                        #IEC_Timer.Spülen(IN := #Zst."TON_CM05.QM62_auf" AND #Out.QM63,
                                          PT := #Param.Spülzeit,
                                          Q => #Zst.Spuelen,
                                          ET => #Spülzeit);
                        #Zst.Restzeit_Spülen := #Param.Spülzeit - #Spülzeit;

                        IF #Zst."TON_CM05.QM62_auf" AND #Out.QM63 AND #In."SRM_CM05.QM61_zu" AND #In."SRM_CM05.QM64_zu" AND NOT #Zst.Spuelen THEN
                            #Zst.Spuelen_aktiv := FALSE;
                            #Out.QM62 := FALSE;
                        END_IF;

                        // Fertig
                        IF NOT #Zst.Spuelen AND NOT #Zst.Spuelen_aktiv AND NOT #Out.QM63 THEN
                            #Out.QM62 := #Out.QM63 := FALSE;
                            #Zst.Restzeit_Spülen := T#0s;
                            #Mld.Pu_Spuelen_Fertig := TRUE;
                        END_IF;
                    ELSE
                        #Out.QM62 := FALSE;
                        #Out.QM63 := FALSE;
                        #Zst.Restzeit_Spülen := T#0s;
                    END_IF;
                    #Out.GP11_Ein := FALSE;

           2: // Spülen + Drucktest - nur Hand
               // Ventile Abpumpen zu    
               #Out.QM61 := FALSE;
               #Out.QM64 := FALSE;
               IF NOT #Zst.Drucktest_aktiv THEN
                   IF #In.Ein THEN
                       IF #posFl_Hand THEN
                           #Zst.Spuelen_aktiv := TRUE;
                       END_IF;
                       #Out.QM62 := NOT #In."Niv_max_CM05.BL01" AND NOT #In."Niv_Uel_CM05.BL05";
                       #Out.QM63 := #Out.QM62;
                       #IEC_Timer.Spülen(IN := #Zst."TON_CM05.QM62_auf" AND #Out.QM63 AND #In."SRM_CM05.QM61_zu" AND #In."SRM_CM05.QM64_zu",
                                         PT := #Param.Spülzeit,
                                         Q => #Zst.Spuelen,
                                         ET => #Spülzeit);
                       #Zst.Restzeit_Spülen := #Param.Spülzeit - #Spülzeit;

                       IF #Zst."TON_CM05.QM62_auf" AND #Out.QM63 AND #In."SRM_CM05.QM61_zu" AND #In."SRM_CM05.QM64_zu" AND NOT #Zst.Spuelen THEN
                           #Zst.Spuelen_aktiv := FALSE;
                       END_IF;

                       // Fertig
                       IF NOT #Zst.Spuelen AND NOT #Zst.Spuelen_aktiv THEN
                           #Out.QM62 := #Out.QM63 := FALSE;
                           #Zst.Restzeit_Spülen := T#0s;
                           #Zst.Drucktest_aktiv := TRUE;
                           #Zst.Status_DT := #S1;
                       END_IF;
                   ELSE
                       #Out.QM62 := FALSE;
                       #Out.QM63 := FALSE;
                       #Zst.Restzeit_Spülen := T#0s;
                   END_IF;
                   #Out.GP11_Ein := FALSE;
               END_IF;

               IF #Zst.Drucktest_aktiv THEN
                   CASE #Zst.Status_DT OF
                       #S1:  //Druckaufbau

                           IF "DB_Temporaer".Drucksensoren_deaktiviert THEN
                               #Zst.Drucktest_ok := TRUE;

                               "Ergebnis_DT"("Name" := #"Name",
                                             akt_Zeit := "Uhrzeit".aktDatum,
                                             ok := #Zst.Drucktest_ok,
                                             Fehler := NOT #Zst.Drucktest_ok);

                               #Mld.Drucktest_ok := #Zst.Drucktest_ok;
                               #Mld.DT_Fehler := NOT #Zst.Drucktest_ok;
                               #Zst.Status_DT := #S4;
                           ELSE
                               #Out.QM62 := TRUE;
                               IF (#In.Druck_Pumpe > #Param.SW_Drucktest + 0.25) OR #Mld.TO_Druckaufbau THEN
                                   #Zst.Status_DT := #S2;
                               END_IF;
                               #Zst.Restzeit_DT := #Param.DT_Druckaufbau - #IEC_Timer.TO_Druckaufbau.ET;
                           END_IF;

                       #S2: //Wartezeit
                           #IEC_Timer.Drucktest(IN := NOT #Out.QM62,
                                                PT := #Param.DT_Testzeit,
                                                Q => #Zst.Zeit_laeuft,
                                                ET => #Zeit_DT);
                           #Zst.Restzeit_DT := #Param.DT_Testzeit - #Zeit_DT;

                           IF NOT #Zst.Zeit_laeuft AND NOT #Out.QM62 THEN
                               #Zst.Restzeit_DT := T#0s;
                               #Zst.Status_DT := #S3;
                           END_IF;
                           #Out.QM62 := FALSE;

                       #S3:// Überprüfung
                           #Zst.Drucktest_ok := #In.Druck_Pumpe >= #Param.SW_Drucktest;

                           "Ergebnis_DT"("Name" := #"Name",
                                         akt_Zeit := "Uhrzeit".aktDatum,
                                         ok := #Zst.Drucktest_ok,
                                         Fehler := NOT #Zst.Drucktest_ok);

                           #Mld.Drucktest_ok := #Zst.Drucktest_ok;
                           #Mld.DT_Fehler := NOT #Zst.Drucktest_ok;
                           #Zst.Status_DT := #S4;

                       #S4: // Ende
                           ;
                   END_CASE;
               END_IF;
       END_CASE;
   ELSE
       #Out.GP11_Ein := FALSE;
       #Out.QM61 := FALSE;
       #Out.QM62 := FALSE;
       #Out.QM63 := FALSE;
       #Out.QM64 := FALSE;
   END_IF;
END_REGION

REGION Network 3 (SCL): Überwachung / Meldungen
   // Motorschutzschalter
   #Mld.MSS := NOT #In.MSS_ok AND NOT #In.NotHalt;
   // Trockenlaufschutz
   #Mld."TLS_CM05.BL03" := NOT #In."Niv_TLS_CM05.BL03";
   // Überlauf
   #Mld."Uel_CM05.BL05" := #In."Niv_Uel_CM05.BL05";
   // AWA nicht betriebsbereit
   #Mld.AWA_niO := NOT #In.AWA_ok;
   // keine Freigabe Abpumpen
   #Mld.keine_Frg_AWA := NOT #In.Frg_AWA;

   // Zeitüberschreitung Druckaufbau
   #IEC_Timer.TO_Druckaufbau(IN := #Zst.Status_DT = #S1,
                             PT := #Param.DT_Druckaufbau,
                             Q => #Mld.TO_Druckaufbau);

   // Grenzwert Pumpendruck
   #IEC_Timer.GW_p(IN := #Out.GP11_Ein,
                   PT := T#3s,
                   Q => #GP11_Laeuft);

   #Mld.GW_p := #GP11_Laeuft AND #In.GW_p;
   // nicht in Automatik
   #Mld.n_Auto := NOT #In.Auto AND "DB_ANLAGE".BA.Automat_ein;
END_REGION

REGION Network 4 (SCL): --> Visu
   // Status Pumpe
   "Status_E0A"(Hand := #In.Ein,
                Auto := #In.Auto,
                SonderModus_PumpeSpuelen:=#Zst.Spuelen,
                Stoerung := NOT #In.MSS_ok,
                Ausgang := #Out.GP11_Ein,
                StatusByte => #Zst.Status_GP11);
   // Anzeige Füllstand
   "Niv_Visu"(Niv_1 := #In."Niv_TLS_CM05.BL03",
              Niv_2 := #In."Niv_min_CM05.BL02",
              Niv_3 := #In."Niv_max_CM05.BL01",
              Niv_4 := #In."Niv_Uel_CM05.BL05",
              Niv_5 := FALSE,
              Niv_6 := FALSE,
              Wert_1 := #Niv_TLS,
              Wert_2 := #Niv_Min,
              Wert_3 := #Niv_max,
              Wert_4 := #Niv_Uel,
              Wert_5 := 0,
              Wert_6 := 0,
              Niveau => #Zst.Niveau,
              Niv_Err => #Mld.Niv_Sensorfehler);
END_REGION
END_FUNCTION_BLOCK

FUNCTION_BLOCK "Ventil_Stati"   // FB1095, LAD
TITLE = Ventilstatus
{ S7_Optimized_Access := 'TRUE' }
// 0: geschlossen (grau)
// 1: geöffnet (grün)
// 2: Störung (rot)
// stored: AutoNumber false, MemoryReserve 100, SetENOAutomatically false
   VAR RETAIN
      Param { ExternalAccessible := 'False'; ExternalVisible := 'False'; ExternalWritable := 'False'} : Struct
         "TO" : Time := T#20s;
      END_STRUCT;
      Mld : Struct
         "TO_auf_CM01.QM18" : Bool;
         "TO_zu_CM01.QM18" : Bool;
         "SF_CM01.QM18" : Bool;
         "TO_auf_CM01.QM19" : Bool;
         "TO_zu_CM01.QM19" : Bool;
         "SF_CM01.QM19" : Bool;
         "TO_auf_CM01.QM20" : Bool;
         "TO_zu_CM01.QM20" : Bool;
         "SF_CM01.QM20" : Bool;
         "TO_auf_CM01.QM25" : Bool;
         "TO_zu_CM01.QM25" : Bool;
         "SF_CM01.QM25" : Bool;
         "TO_auf_CM01.QM26" : Bool;
         "TO_zu_CM01.QM26" : Bool;
         "SF_CM01.QM26" : Bool;
         "TO_auf_CM01.QM27" : Bool;
         "TO_zu_CM01.QM27" : Bool;
         "SF_CM01.QM27" : Bool;
         "TO_auf_CM02.QM55" : Bool;
         "TO_zu_CM02.QM55" : Bool;
         "SF_CM02.QM55" : Bool;
         "TO_auf_CM02.QM56" : Bool;
         "TO_zu_CM02.QM56" : Bool;
         "SF_CM02.QM56" : Bool;
         "TO_auf_CM02.QM57" : Bool;
         "TO_zu_CM02.QM57" : Bool;
         "SF_CM02.QM57" : Bool;
         "TO_auf_CM02.QM62" : Bool;
         "TO_zu_CM02.QM62" : Bool;
         "SF_CM02.QM62" : Bool;
         "TO_auf_CM02.QM63" : Bool;
         "TO_zu_CM02.QM63" : Bool;
         "SF_CM02.QM63" : Bool;
         "TO_auf_CM02.QM64" : Bool;
         "TO_zu_CM02.QM64" : Bool;
         "SF_CM02.QM64" : Bool;
         "TO_auf_HQ01.QM21" : Bool;
         "TO_zu_HQ01.QM21" : Bool;
         "SF_HQ01.QM21" : Bool;
         "TO_auf_HQ01.QM22" : Bool;
         "TO_zu_HQ01.QM22" : Bool;
         "SF_HQ01.QM22" : Bool;
         "TO_auf_HQ01.QM23" : Bool;
         "TO_zu_HQ01.QM23" : Bool;
         "SF_HQ01.QM23" : Bool;
         "TO_auf_HQ01.QM24" : Bool;
         "TO_zu_HQ01.QM24" : Bool;
         "SF_HQ01.QM24" : Bool;
         "TO_auf_HQ01.LV01" : Bool;
         "TO_zu_HQ01.LV01" : Bool;
         "SF_HQ01.LV01" : Bool;
         "TO_auf_HQ02.QM58" : Bool;
         "TO_zu_HQ02.QM58" : Bool;
         "SF_HQ02.QM58" : Bool;
         "TO_auf_HQ02.QM59" : Bool;
         "TO_zu_HQ02.QM59" : Bool;
         "SF_HQ02.QM59" : Bool;
         "TO_auf_HQ02.QM60" : Bool;
         "TO_zu_HQ02.QM60" : Bool;
         "SF_HQ02.QM60" : Bool;
         "TO_auf_HQ02.QM61" : Bool;
         "TO_zu_HQ02.QM61" : Bool;
         "SF_HQ02.QM61" : Bool;
         "TO_auf_HQ02.LV02" : Bool;
         "TO_zu_HQ02.LV02" : Bool;
         "SF_HQ02.LV02" : Bool;
         "TO_auf_CM03.QM33" : Bool;
         "TO_zu_CM03.QM33" : Bool;
         "SF_CM03.QM33" : Bool;
         "TO_auf_CM03.QM34" : Bool;
         "TO_zu_CM03.QM34" : Bool;
         "SF_CM03.QM34" : Bool;
         "TO_auf_CM04.QM72" : Bool;
         "TO_zu_CM04.QM72" : Bool;
         "SF_CM04.QM72" : Bool;
         "TO_auf_CM04.QM73" : Bool;
         "TO_zu_CM04.QM73" : Bool;
         "SF_CM04.QM73" : Bool;
         "TO_auf_CM05.QM61" : Bool;
         "TO_zu_CM05.QM61" : Bool;
         "SF_CM05.QM61" : Bool;
         "TO_auf_CM05.QM64" : Bool;
         "TO_zu_CM05.QM64" : Bool;
         "SF_CM05.QM64" : Bool;
         "TO_auf_GP01.QM14" : Bool;
         "TO_zu_GP01.QM14" : Bool;
         "SF_GP01.QM14" : Bool;
         "TO_auf_GP01.QM15" : Bool;
         "TO_zu_GP01.QM15" : Bool;
         "SF_GP01.QM15" : Bool;
         "TO_auf_GP01.QM16" : Bool;
         "TO_zu_GP01.QM16" : Bool;
         "SF_GP01.QM16" : Bool;
         "TO_auf_GP01.QM17" : Bool;
         "TO_zu_GP01.QM17" : Bool;
         "SF_GP01.QM17" : Bool;
         "TO_auf_GP01.QM18" : Bool;
         "TO_zu_GP01.QM18" : Bool;
         "SF_GP01.QM18" : Bool;
         "TO_auf_GP01.QM19" : Bool;
         "TO_zu_GP01.QM19" : Bool;
         "SF_GP01.QM19" : Bool;
         "TO_auf_GP01.QM20" : Bool;
         "TO_zu_GP01.QM20" : Bool;
         "SF_GP01.QM20" : Bool;
         "TO_auf_GP01.QM21" : Bool;
         "TO_zu_GP01.QM21" : Bool;
         "SF_GP01.QM21" : Bool;
         "TO_auf_GP01.QM22" : Bool;
         "TO_zu_GP01.QM22" : Bool;
         "SF_GP01.QM22" : Bool;
         "TO_auf_GP02.QM38" : Bool;
         "TO_zu_GP02.QM38" : Bool;
         "SF_GP02.QM38" : Bool;
         "TO_auf_GP02.QM39" : Bool;
         "TO_zu_GP02.QM39" : Bool;
         "SF_GP02.QM39" : Bool;
         "TO_auf_GP02.QM40" : Bool;
         "TO_zu_GP02.QM40" : Bool;
         "SF_GP02.QM40" : Bool;
         "TO_auf_GP02.QM41" : Bool;
         "TO_zu_GP02.QM41" : Bool;
         "SF_GP02.QM41" : Bool;
         "TO_auf_GP02.QM42" : Bool;
         "TO_zu_GP02.QM42" : Bool;
         "SF_GP02.QM42" : Bool;
         "TO_auf_GP02.QM43" : Bool;
         "TO_zu_GP02.QM43" : Bool;
         "SF_GP02.QM43" : Bool;
         "TO_auf_GP02.QM44" : Bool;
         "TO_zu_GP02.QM44" : Bool;
         "SF_GP02.QM44" : Bool;
         "TO_auf_GP02.QM45" : Bool;
         "TO_zu_GP02.QM45" : Bool;
         "SF_GP02.QM45" : Bool;
         "TO_auf_GP02.QM46" : Bool;
         "TO_zu_GP02.QM46" : Bool;
         "SF_GP02.QM46" : Bool;
      END_STRUCT;
   END_VAR
   VAR
      IEC_Timer { ExternalAccessible := 'False'; ExternalVisible := 'False'; ExternalWritable := 'False'} : Struct
         "TO_auf_CM01.QM18" { S7_SetPoint := 'True'} : TON_TIME;
         "TO_zu_CM01.QM18" { S7_SetPoint := 'True'} : TON_TIME;
         "TO_auf_CM01.QM19" { S7_SetPoint := 'True'} : TON_TIME;
         "TO_zu_CM01.QM19" { S7_SetPoint := 'True'} : TON_TIME;
         "TO_auf_CM01.QM20" { S7_SetPoint := 'True'} : TON_TIME;
         "TO_zu_CM01.QM20" { S7_SetPoint := 'True'} : TON_TIME;
         "TO_auf_CM01.QM25" { S7_SetPoint := 'True'} : TON_TIME;
         "TO_zu_CM01.QM25" { S7_SetPoint := 'True'} : TON_TIME;
         "TO_auf_CM01.QM26" { S7_SetPoint := 'True'} : TON_TIME;
         "TO_zu_CM01.QM26" { S7_SetPoint := 'True'} : TON_TIME;
         "TO_auf_CM01.QM27" { S7_SetPoint := 'True'} : TON_TIME;
         "TO_zu_CM01.QM27" { S7_SetPoint := 'True'} : TON_TIME;
         "TO_auf_CM02.QM55" { S7_SetPoint := 'True'} : TON_TIME;
         "TO_zu_CM02.QM55" { S7_SetPoint := 'True'} : TON_TIME;
         "TO_auf_CM02.QM56" { S7_SetPoint := 'True'} : TON_TIME;
         "TO_zu_CM02.QM56" { S7_SetPoint := 'True'} : TON_TIME;
         "TO_auf_CM02.QM57" { S7_SetPoint := 'True'} : TON_TIME;
         "TO_zu_CM02.QM57" { S7_SetPoint := 'True'} : TON_TIME;
         "TO_auf_CM02.QM62" { S7_SetPoint := 'True'} : TON_TIME;
         "TO_zu_CM02.QM62" { S7_SetPoint := 'True'} : TON_TIME;
         "TO_auf_CM02.QM63" { S7_SetPoint := 'True'} : TON_TIME;
         "TO_zu_CM02.QM63" { S7_SetPoint := 'True'} : TON_TIME;
         "TO_auf_CM02.QM64" { S7_SetPoint := 'True'} : TON_TIME;
         "TO_zu_CM02.QM64" { S7_SetPoint := 'True'} : TON_TIME;
         "TO_auf_HQ01.QM21" { S7_SetPoint := 'True'} : TON_TIME;
         "TO_zu_HQ01.QM21" { S7_SetPoint := 'True'} : TON_TIME;
         "TO_auf_HQ01.QM22" { S7_SetPoint := 'True'} : TON_TIME;
         "TO_zu_HQ01.QM22" { S7_SetPoint := 'True'} : TON_TIME;
         "TO_auf_HQ01.QM23" { S7_SetPoint := 'True'} : TON_TIME;
         "TO_zu_HQ01.QM23" { S7_SetPoint := 'True'} : TON_TIME;
         "TO_auf_HQ01.QM24" { S7_SetPoint := 'True'} : TON_TIME;
         "TO_zu_HQ01.QM24" { S7_SetPoint := 'True'} : TON_TIME;
         "TO_auf_HQ01.LV01" { S7_SetPoint := 'True'} : TON_TIME;
         "TO_zu_HQ01.LV01" { S7_SetPoint := 'True'} : TON_TIME;
         "TO_auf_HQ02.QM58" { S7_SetPoint := 'True'} : TON_TIME;
         "TO_zu_HQ02.QM58" { S7_SetPoint := 'True'} : TON_TIME;
         "TO_auf_HQ02.QM59" { S7_SetPoint := 'True'} : TON_TIME;
         "TO_zu_HQ02.QM59" { S7_SetPoint := 'True'} : TON_TIME;
         "TO_auf_HQ02.QM60" { S7_SetPoint := 'True'} : TON_TIME;
         "TO_zu_HQ02.QM60" { S7_SetPoint := 'True'} : TON_TIME;
         "TO_auf_HQ02.QM61" { S7_SetPoint := 'True'} : TON_TIME;
         "TO_zu_HQ02.QM61" { S7_SetPoint := 'True'} : TON_TIME;
         "TO_auf_HQ02.LV02" { S7_SetPoint := 'True'} : TON_TIME;
         "TO_zu_HQ02.LV02" { S7_SetPoint := 'True'} : TON_TIME;
         "TO_auf_CM03.QM33" { S7_SetPoint := 'True'} : TON_TIME;
         "TO_zu_CM03.QM33" { S7_SetPoint := 'True'} : TON_TIME;
         "TO_auf_CM03.QM34" { S7_SetPoint := 'True'} : TON_TIME;
         "TO_zu_CM03.QM34" { S7_SetPoint := 'True'} : TON_TIME;
         "TO_auf_CM04.QM72" { S7_SetPoint := 'True'} : TON_TIME;
         "TO_zu_CM04.QM72" { S7_SetPoint := 'True'} : TON_TIME;
         "TO_auf_CM04.QM73" { S7_SetPoint := 'True'} : TON_TIME;
         "TO_zu_CM04.QM73" { S7_SetPoint := 'True'} : TON_TIME;
         "TO_auf_CM05.QM61" { S7_SetPoint := 'True'} : TON_TIME;
         "TO_zu_CM05.QM61" { S7_SetPoint := 'True'} : TON_TIME;
         "TO_auf_CM05.QM64" { S7_SetPoint := 'True'} : TON_TIME;
         "TO_zu_CM05.QM64" { S7_SetPoint := 'True'} : TON_TIME;
         "TO_auf_GP01.QM14" { S7_SetPoint := 'True'} : TON_TIME;
         "TO_zu_GP01.QM14" { S7_SetPoint := 'True'} : TON_TIME;
         "TO_auf_GP01.QM15" { S7_SetPoint := 'True'} : TON_TIME;
         "TO_zu_GP01.QM15" { S7_SetPoint := 'True'} : TON_TIME;
         "TO_auf_GP01.QM16" { S7_SetPoint := 'True'} : TON_TIME;
         "TO_zu_GP01.QM16" { S7_SetPoint := 'True'} : TON_TIME;
         "TO_auf_GP01.QM17" { S7_SetPoint := 'True'} : TON_TIME;
         "TO_zu_GP01.QM17" { S7_SetPoint := 'True'} : TON_TIME;
         "TO_auf_GP01.QM18" { S7_SetPoint := 'True'} : TON_TIME;
         "TO_zu_GP01.QM18" { S7_SetPoint := 'True'} : TON_TIME;
         "TO_auf_GP01.QM19" { S7_SetPoint := 'True'} : TON_TIME;
         "TO_zu_GP01.QM19" { S7_SetPoint := 'True'} : TON_TIME;
         "TO_auf_GP01.QM20" { S7_SetPoint := 'True'} : TON_TIME;
         "TO_zu_GP01.QM20" { S7_SetPoint := 'True'} : TON_TIME;
         "TO_auf_GP01.QM21" { S7_SetPoint := 'True'} : TON_TIME;
         "TO_zu_GP01.QM21" { S7_SetPoint := 'True'} : TON_TIME;
         "TO_auf_GP01.QM22" { S7_SetPoint := 'True'} : TON_TIME;
         "TO_zu_GP01.QM22" { S7_SetPoint := 'True'} : TON_TIME;
         "TO_auf_GP02.QM38" { S7_SetPoint := 'True'} : TON_TIME;
         "TO_zu_GP02.QM38" { S7_SetPoint := 'True'} : TON_TIME;
         "TO_auf_GP02.QM39" { S7_SetPoint := 'True'} : TON_TIME;
         "TO_zu_GP02.QM39" { S7_SetPoint := 'True'} : TON_TIME;
         "TO_auf_GP02.QM40" { S7_SetPoint := 'True'} : TON_TIME;
         "TO_zu_GP02.QM40" { S7_SetPoint := 'True'} : TON_TIME;
         "TO_auf_GP02.QM41" { S7_SetPoint := 'True'} : TON_TIME;
         "TO_zu_GP02.QM41" { S7_SetPoint := 'True'} : TON_TIME;
         "TO_auf_GP02.QM42" { S7_SetPoint := 'True'} : TON_TIME;
         "TO_zu_GP02.QM42" { S7_SetPoint := 'True'} : TON_TIME;
         "TO_auf_GP02.QM43" { S7_SetPoint := 'True'} : TON_TIME;
         "TO_zu_GP02.QM43" { S7_SetPoint := 'True'} : TON_TIME;
         "TO_auf_GP02.QM44" { S7_SetPoint := 'True'} : TON_TIME;
         "TO_zu_GP02.QM44" { S7_SetPoint := 'True'} : TON_TIME;
         "TO_auf_GP02.QM45" { S7_SetPoint := 'True'} : TON_TIME;
         "TO_zu_GP02.QM45" { S7_SetPoint := 'True'} : TON_TIME;
         "TO_auf_GP02.QM46" { S7_SetPoint := 'True'} : TON_TIME;
         "TO_zu_GP02.QM46" { S7_SetPoint := 'True'} : TON_TIME;
      END_STRUCT;
   END_VAR
   VAR CONSTANT
      grau : USInt;
      grün : USInt := 1;
      rot : USInt := 2;
   END_VAR
BEGIN

REGION Network 1 (SCL): CM01

   "Ventilstatus"(SRM_auf:= "E_SRM_CM01.QM18_auf",
                  SRM_zu:= "E_SRM_CM01.QM18_zu",
                  A_Ventil:= "A_CM01.QM18",
                  Zeit:= #Param.TO,
                  "Farbe HMI"=> "Panel".Ventil."CM01.QM18",
                  Mld_Sensorfehler:= #Mld."SF_CM01.QM18",
                  Mld_TO_oeffnen=> #Mld."TO_auf_CM01.QM18",
                  Mld_TO_schliessen=> #Mld."TO_zu_CM01.QM18",
                  TO_oeffnen:= #IEC_Timer."TO_auf_CM01.QM18",
                  TO_schliessen:= #IEC_Timer."TO_zu_CM01.QM18");

   "Ventilstatus"(SRM_auf := "E_SRM_CM01.QM19_auf",
                  SRM_zu := "E_SRM_CM01.QM19_zu",
                  A_Ventil := "A_CM01.QM19",
                  Zeit := #Param.TO,
                  "Farbe HMI" => "Panel".Ventil."CM01.QM19",
                  Mld_Sensorfehler := #Mld."SF_CM01.QM19",
                  Mld_TO_oeffnen => #Mld."TO_auf_CM01.QM19",
                  Mld_TO_schliessen => #Mld."TO_zu_CM01.QM19",
                  TO_oeffnen := #IEC_Timer."TO_auf_CM01.QM19",
                  TO_schliessen := #IEC_Timer."TO_zu_CM01.QM19");

   "Ventilstatus"(SRM_auf := "E_SRM_CM01.QM20_auf",
                  SRM_zu := "E_SRM_CM01.QM20_zu",
                  A_Ventil := "A_CM01.QM20",
                  Zeit := #Param.TO,
                  "Farbe HMI" => "Panel".Ventil."CM01.QM20",
                  Mld_Sensorfehler := #Mld."SF_CM01.QM20",
                  Mld_TO_oeffnen => #Mld."TO_auf_CM01.QM20",
                  Mld_TO_schliessen => #Mld."TO_zu_CM01.QM20",
                  TO_oeffnen := #IEC_Timer."TO_auf_CM01.QM20",
                  TO_schliessen := #IEC_Timer."TO_zu_CM01.QM20");

   "Ventilstatus"(SRM_auf := "E_SRM_CM01.QM25_auf",
                  SRM_zu := "E_SRM_CM01.QM25_zu",
                  A_Ventil := "A_CM01.QM25",
                  Zeit := #Param.TO,
                  "Farbe HMI" => "Panel".Ventil."CM01.QM25",
                  Mld_Sensorfehler := #Mld."SF_CM01.QM25",
                  Mld_TO_oeffnen => #Mld."TO_auf_CM01.QM25",
                  Mld_TO_schliessen => #Mld."TO_zu_CM01.QM25",
                  TO_oeffnen := #IEC_Timer."TO_auf_CM01.QM25",
                  TO_schliessen := #IEC_Timer."TO_zu_CM01.QM25");

   "Ventilstatus"(SRM_auf := "E_SRM_CM01.QM26_auf",
                  SRM_zu := "E_SRM_CM01.QM26_zu",
                  A_Ventil := "A_CM01.QM26",
                  Zeit := #Param.TO,
                  "Farbe HMI" => "Panel".Ventil."CM01.QM26",
                  Mld_Sensorfehler := #Mld."SF_CM01.QM26",
                  Mld_TO_oeffnen => #Mld."TO_auf_CM01.QM26",
                  Mld_TO_schliessen => #Mld."TO_zu_CM01.QM26",
                  TO_oeffnen := #IEC_Timer."TO_auf_CM01.QM26",
                  TO_schliessen := #IEC_Timer."TO_zu_CM01.QM26");

   "Ventilstatus"(SRM_auf := "E_SRM_CM01.QM27_auf",
                  SRM_zu := "E_SRM_CM01.QM27_zu",
                  A_Ventil := "A_CM01.QM27",
                  Zeit := #Param.TO,
                  "Farbe HMI" => "Panel".Ventil."CM01.QM27",
                  Mld_Sensorfehler := #Mld."SF_CM01.QM27",
                  Mld_TO_oeffnen => #Mld."TO_auf_CM01.QM27",
                  Mld_TO_schliessen => #Mld."TO_zu_CM01.QM27",
                  TO_oeffnen := #IEC_Timer."TO_auf_CM01.QM27",
                  TO_schliessen := #IEC_Timer."TO_zu_CM01.QM27");
END_REGION

REGION Network 2 (SCL): HQ01
   "Ventilstatus"(SRM_auf := "E_SRM_HQ01.LV01_auf",
                  SRM_zu := "E_SRM_HQ01.LV01_zu",
                  A_Ventil := "A_HQ01.LV01",
                  Zeit := #Param.TO,
                  "Farbe HMI" => "Panel".Ventil."HQ01.LV01",
                  Mld_Sensorfehler := #Mld."SF_HQ01.LV01",
                  Mld_TO_oeffnen => #Mld."TO_auf_HQ01.LV01",
                  Mld_TO_schliessen => #Mld."TO_zu_HQ01.LV01",
                  TO_oeffnen := #IEC_Timer."TO_auf_HQ01.LV01",
                  TO_schliessen := #IEC_Timer."TO_zu_HQ01.LV01");

   "Ventilstatus"(SRM_auf := "E_SRM_HQ01.QM21_auf",
                  SRM_zu := "E_SRM_HQ01.QM21_zu",
                  A_Ventil := "A_HQ01.QM21",
                  Zeit := #Param.TO,
                  "Farbe HMI" => "Panel".Ventil."HQ01.QM21",
                  Mld_Sensorfehler := #Mld."SF_HQ01.QM21",
                  Mld_TO_oeffnen => #Mld."TO_auf_HQ01.QM21",
                  Mld_TO_schliessen => #Mld."TO_zu_HQ01.QM21",
                  TO_oeffnen := #IEC_Timer."TO_auf_HQ01.QM21",
                  TO_schliessen := #IEC_Timer."TO_zu_HQ01.QM21");

   "Ventilstatus"(SRM_auf := "E_SRM_HQ01.QM22_auf",
                  SRM_zu := "E_SRM_HQ01.QM22_zu",
                  A_Ventil := "A_HQ01.QM22",
                  Zeit := #Param.TO,
                  "Farbe HMI" => "Panel".Ventil."HQ01.QM22",
                  Mld_Sensorfehler := #Mld."SF_HQ01.QM22",
                  Mld_TO_oeffnen => #Mld."TO_auf_HQ01.QM22",
                  Mld_TO_schliessen => #Mld."TO_zu_HQ01.QM22",
                  TO_oeffnen := #IEC_Timer."TO_auf_HQ01.QM22",
                  TO_schliessen := #IEC_Timer."TO_zu_HQ01.QM22");

   "Ventilstatus"(SRM_auf := "E_SRM_HQ01.QM23_auf",
                  SRM_zu := "E_SRM_HQ01.QM23_zu",
                  A_Ventil := "A_HQ01.QM23",
                  Zeit := #Param.TO,
                  "Farbe HMI" => "Panel".Ventil."HQ01.QM23",
                  Mld_Sensorfehler := #Mld."SF_HQ01.QM23",
                  Mld_TO_oeffnen => #Mld."TO_auf_HQ01.QM23",
                  Mld_TO_schliessen => #Mld."TO_zu_HQ01.QM23",
                  TO_oeffnen := #IEC_Timer."TO_auf_HQ01.QM23",
                  TO_schliessen := #IEC_Timer."TO_zu_HQ01.QM23");

   "Ventilstatus"(SRM_auf := "E_SRM_HQ01.QM24_auf",
                  SRM_zu := "E_SRM_HQ01.QM24_zu",
                  A_Ventil := "A_HQ01.QM24",
                  Zeit := #Param.TO,
                  "Farbe HMI" => "Panel".Ventil."HQ01.QM24",
                  Mld_Sensorfehler := #Mld."SF_HQ01.QM24",
                  Mld_TO_oeffnen => #Mld."TO_auf_HQ01.QM24",
                  Mld_TO_schliessen => #Mld."TO_zu_HQ01.QM24",
                  TO_oeffnen := #IEC_Timer."TO_auf_HQ01.QM24",
                  TO_schliessen := #IEC_Timer."TO_zu_HQ01.QM24");
END_REGION

REGION Network 3 (SCL): CM03

   "Ventilstatus"(SRM_auf := "E_SRM_CM03.QM33_auf",
                  SRM_zu := "E_SRM_CM03.QM33_zu",
                  A_Ventil := "A_CM03.QM33",
                  Zeit := #Param.TO,
                  "Farbe HMI" => "Panel".Ventil."CM03.QM33",
                  Mld_Sensorfehler := #Mld."SF_CM03.QM33",
                  Mld_TO_oeffnen => #Mld."TO_auf_CM03.QM33",
                  Mld_TO_schliessen => #Mld."TO_zu_CM03.QM33",
                  TO_oeffnen := #IEC_Timer."TO_auf_CM03.QM33",
                  TO_schliessen := #IEC_Timer."TO_zu_CM03.QM33");

   "Ventilstatus"(SRM_auf := "E_SRM_CM03.QM34_auf",
                  SRM_zu := "E_SRM_CM03.QM34_zu",
                  A_Ventil := "A_CM03.QM34",
                  Zeit := #Param.TO,
                  "Farbe HMI" => "Panel".Ventil."CM03.QM34",
                  Mld_Sensorfehler := #Mld."SF_CM03.QM34",
                  Mld_TO_oeffnen => #Mld."TO_auf_CM03.QM34",
                  Mld_TO_schliessen => #Mld."TO_zu_CM03.QM34",
                  TO_oeffnen := #IEC_Timer."TO_auf_CM03.QM34",
                  TO_schliessen := #IEC_Timer."TO_zu_CM03.QM34");

   "Ventilstatus_einfach"(A_Ventil:="A_CM03.QM35",
                          "Farbe HMI"=>"Panel".Ventil."CM03.QM35");

   "Ventilstatus_einfach"(A_Ventil := "A_CM03.QM36",
                          "Farbe HMI" => "Panel".Ventil."CM03.QM36");

   "Ventilstatus_einfach"(A_Ventil := "A_CM03.QM37",
                          "Farbe HMI" => "Panel".Ventil."CM03.QM37");
END_REGION

REGION Network 4 (SCL): CM02

   "Ventilstatus"(SRM_auf := "E_SRM_CM02.QM55_auf",
                  SRM_zu := "E_SRM_CM02.QM55_zu",
                  A_Ventil := "A_CM02.QM55",
                  Zeit := #Param.TO,
                  "Farbe HMI" => "Panel".Ventil."CM02.QM55",
                  Mld_Sensorfehler := #Mld."SF_CM02.QM55",
                  Mld_TO_oeffnen => #Mld."TO_auf_CM02.QM55",
                  Mld_TO_schliessen => #Mld."TO_zu_CM02.QM55",
                  TO_oeffnen := #IEC_Timer."TO_auf_CM02.QM55",
                  TO_schliessen := #IEC_Timer."TO_zu_CM02.QM55");

   "Ventilstatus"(SRM_auf := "E_SRM_CM02.QM56_auf",
                  SRM_zu := "E_SRM_CM02.QM56_zu",
                  A_Ventil := "A_CM02.QM56",
                  Zeit := #Param.TO,
                  "Farbe HMI" => "Panel".Ventil."CM02.QM56",
                  Mld_Sensorfehler := #Mld."SF_CM02.QM56",
                  Mld_TO_oeffnen => #Mld."TO_auf_CM02.QM56",
                  Mld_TO_schliessen => #Mld."TO_zu_CM02.QM56",
                  TO_oeffnen := #IEC_Timer."TO_auf_CM02.QM56",
                  TO_schliessen := #IEC_Timer."TO_zu_CM02.QM56");

   "Ventilstatus"(SRM_auf := "E_SRM_CM02.QM57_auf",
                  SRM_zu := "E_SRM_CM02.QM57_zu",
                  A_Ventil := "A_CM02.QM57",
                  Zeit := #Param.TO,
                  "Farbe HMI" => "Panel".Ventil."CM02.QM57",
                  Mld_Sensorfehler := #Mld."SF_CM02.QM57",
                  Mld_TO_oeffnen => #Mld."TO_auf_CM02.QM57",
                  Mld_TO_schliessen => #Mld."TO_zu_CM02.QM57",
                  TO_oeffnen := #IEC_Timer."TO_auf_CM02.QM57",
                  TO_schliessen := #IEC_Timer."TO_zu_CM02.QM57");

   "Ventilstatus"(SRM_auf := "E_SRM_CM02.QM62_auf",
                  SRM_zu := "E_SRM_CM02.QM62_zu",
                  A_Ventil := "A_CM02.QM62",
                  Zeit := #Param.TO,
                  "Farbe HMI" => "Panel".Ventil."CM02.QM62",
                  Mld_Sensorfehler := #Mld."SF_CM02.QM62",
                  Mld_TO_oeffnen => #Mld."TO_auf_CM02.QM62",
                  Mld_TO_schliessen => #Mld."TO_zu_CM02.QM62",
                  TO_oeffnen := #IEC_Timer."TO_auf_CM02.QM62",
                  TO_schliessen := #IEC_Timer."TO_zu_CM02.QM62");

   "Ventilstatus"(SRM_auf := "E_SRM_CM02.QM63_auf",
                  SRM_zu := "E_SRM_CM02.QM63_zu",
                  A_Ventil := "A_CM02.QM63",
                  Zeit := #Param.TO,
                  "Farbe HMI" => "Panel".Ventil."CM02.QM63",
                  Mld_Sensorfehler := #Mld."SF_CM02.QM63",
                  Mld_TO_oeffnen => #Mld."TO_auf_CM02.QM63",
                  Mld_TO_schliessen => #Mld."TO_zu_CM02.QM63",
                  TO_oeffnen := #IEC_Timer."TO_auf_CM02.QM63",
                  TO_schliessen := #IEC_Timer."TO_zu_CM02.QM63");

   "Ventilstatus"(SRM_auf := "E_SRM_CM02.QM64_auf",
                  SRM_zu := "E_SRM_CM02.QM64_zu",
                  A_Ventil := "A_CM02.QM64",
                  Zeit := #Param.TO,
                  "Farbe HMI" => "Panel".Ventil."CM02.QM64",
                  Mld_Sensorfehler := #Mld."SF_CM02.QM64",
                  Mld_TO_oeffnen => #Mld."TO_auf_CM02.QM64",
                  Mld_TO_schliessen => #Mld."TO_zu_CM02.QM64",
                  TO_oeffnen := #IEC_Timer."TO_auf_CM02.QM64",
                  TO_schliessen := #IEC_Timer."TO_zu_CM02.QM64");
END_REGION

REGION Network 5 (SCL): HQ02
   "Ventilstatus"(SRM_auf := "E_SRM_HQ02.LV02_auf",
                  SRM_zu := "E_SRM_HQ02.LV02_zu",
                  A_Ventil := "A_HQ02.LV02",
                  Zeit := #Param.TO,
                  "Farbe HMI" => "Panel".Ventil."HQ02.LV02",
                  Mld_Sensorfehler := #Mld."SF_HQ02.LV02",
                  Mld_TO_oeffnen => #Mld."TO_auf_HQ02.LV02",
                  Mld_TO_schliessen => #Mld."TO_zu_HQ02.LV02",
                  TO_oeffnen := #IEC_Timer."TO_auf_HQ02.LV02",
                  TO_schliessen := #IEC_Timer."TO_zu_HQ02.LV02");

   "Ventilstatus"(SRM_auf := "E_SRM_HQ02.QM58_auf",
                  SRM_zu := "E_SRM_HQ02.QM58_zu",
                  A_Ventil := "A_HQ02.QM58",
                  Zeit := #Param.TO,
                  "Farbe HMI" => "Panel".Ventil."HQ02.QM58",
                  Mld_Sensorfehler := #Mld."SF_HQ02.QM58",
                  Mld_TO_oeffnen => #Mld."TO_auf_HQ02.QM58",
                  Mld_TO_schliessen => #Mld."TO_zu_HQ02.QM58",
                  TO_oeffnen := #IEC_Timer."TO_auf_HQ02.QM58",
                  TO_schliessen := #IEC_Timer."TO_zu_HQ02.QM58");

   "Ventilstatus"(SRM_auf := "E_SRM_HQ02.QM59_auf",
                  SRM_zu := "E_SRM_HQ02.QM59_zu",
                  A_Ventil := "A_HQ02.QM59",
                  Zeit := #Param.TO,
                  "Farbe HMI" => "Panel".Ventil."HQ02.QM59",
                  Mld_Sensorfehler := #Mld."SF_HQ02.QM59",
                  Mld_TO_oeffnen => #Mld."TO_auf_HQ02.QM59",
                  Mld_TO_schliessen => #Mld."TO_zu_HQ02.QM59",
                  TO_oeffnen := #IEC_Timer."TO_auf_HQ02.QM59",
                  TO_schliessen := #IEC_Timer."TO_zu_HQ02.QM59");

   "Ventilstatus"(SRM_auf := "E_SRM_HQ02.QM60_auf",
                  SRM_zu := "E_SRM_HQ02.QM60_zu",
                  A_Ventil := "A_HQ02.QM60",
                  Zeit := #Param.TO,
                  "Farbe HMI" => "Panel".Ventil."HQ02.QM60",
                  Mld_Sensorfehler := #Mld."SF_HQ02.QM60",
                  Mld_TO_oeffnen => #Mld."TO_auf_HQ02.QM60",
                  Mld_TO_schliessen => #Mld."TO_zu_HQ02.QM60",
                  TO_oeffnen := #IEC_Timer."TO_auf_HQ02.QM60",
                  TO_schliessen := #IEC_Timer."TO_zu_HQ02.QM60");

   "Ventilstatus"(SRM_auf := "E_SRM_HQ02.QM61_auf",
                  SRM_zu := "E_SRM_HQ02.QM61_zu",
                  A_Ventil := "A_HQ02.QM61",
                  Zeit := #Param.TO,
                  "Farbe HMI" => "Panel".Ventil."HQ02.QM61",
                  Mld_Sensorfehler := #Mld."SF_HQ02.QM61",
                  Mld_TO_oeffnen => #Mld."TO_auf_HQ02.QM61",
                  Mld_TO_schliessen => #Mld."TO_zu_HQ02.QM61",
                  TO_oeffnen := #IEC_Timer."TO_auf_HQ02.QM61",
                  TO_schliessen := #IEC_Timer."TO_zu_HQ02.QM61");
END_REGION

REGION Network 6 (SCL): CM04

   "Ventilstatus"(SRM_auf := "E_SRM_CM04.QM72_auf",
                  SRM_zu := "E_SRM_CM04.QM72_zu",
                  A_Ventil := "A_CM04.QM72",
                  Zeit := #Param.TO,
                  "Farbe HMI" => "Panel".Ventil."CM04.QM72",
                  Mld_Sensorfehler := #Mld."SF_CM04.QM72",
                  Mld_TO_oeffnen => #Mld."TO_auf_CM04.QM72",
                  Mld_TO_schliessen => #Mld."TO_zu_CM04.QM72",
                  TO_oeffnen := #IEC_Timer."TO_auf_CM04.QM72",
                  TO_schliessen := #IEC_Timer."TO_zu_CM04.QM72");

   "Ventilstatus"(SRM_auf := "E_SRM_CM04.QM73_auf",
                  SRM_zu := "E_SRM_CM04.QM73_zu",
                  A_Ventil := "A_CM04.QM73",
                  Zeit := #Param.TO,
                  "Farbe HMI" => "Panel".Ventil."CM04.QM73",
                  Mld_Sensorfehler := #Mld."SF_CM04.QM73",
                  Mld_TO_oeffnen => #Mld."TO_auf_CM04.QM73",
                  Mld_TO_schliessen => #Mld."TO_zu_CM04.QM73",
                  TO_oeffnen := #IEC_Timer."TO_auf_CM04.QM73",
                  TO_schliessen := #IEC_Timer."TO_zu_CM04.QM73");

   "Ventilstatus_einfach"(A_Ventil := "A_CM04.QM74",
                          "Farbe HMI" => "Panel".Ventil."CM04.QM74");

   "Ventilstatus_einfach"(A_Ventil := "A_CM04.QM75",
                          "Farbe HMI" => "Panel".Ventil."CM04.QM75");

   "Ventilstatus_einfach"(A_Ventil := "A_CM04.QM76",
                          "Farbe HMI" => "Panel".Ventil."CM04.QM76");

   "Ventilstatus_einfach"(A_Ventil := "A_CM04.QM77",
                          "Farbe HMI" => "Panel".Ventil."CM04.QM77");
END_REGION

REGION Network 7 (SCL): CM05
   "Ventilstatus"(SRM_auf := "E_SRM_CM05.QM61_auf",
                  SRM_zu := "E_SRM_CM05.QM61_zu",
                  A_Ventil := "A_CM05.QM61",
                  Zeit := #Param.TO,
                  "Farbe HMI" => "Panel".Ventil."CM05.QM61",
                  Mld_Sensorfehler := #Mld."SF_CM05.QM61",
                  Mld_TO_oeffnen => #Mld."TO_auf_CM05.QM61",
                  Mld_TO_schliessen => #Mld."TO_zu_CM05.QM61",
                  TO_oeffnen := #IEC_Timer."TO_auf_CM05.QM61",
                  TO_schliessen := #IEC_Timer."TO_zu_CM05.QM61");

   "Ventilstatus_einfach"(A_Ventil := "A_CM05.QM62",
                          "Farbe HMI" => "Panel".Ventil."CM05.QM62");

   "Ventilstatus_einfach"(A_Ventil := "A_CM05.QM63",
                          "Farbe HMI" => "Panel".Ventil."CM05.QM63");

   "Ventilstatus"(SRM_auf := "E_SRM_CM05.QM64_auf",
                  SRM_zu := "E_SRM_CM05.QM64_zu",
                  A_Ventil := "A_CM05.QM64",
                  Zeit := #Param.TO,
                  "Farbe HMI" => "Panel".Ventil."CM05.QM64",
                  Mld_Sensorfehler := #Mld."SF_CM05.QM64",
                  Mld_TO_oeffnen => #Mld."TO_auf_CM05.QM64",
                  Mld_TO_schliessen => #Mld."TO_zu_CM05.QM64",
                  TO_oeffnen := #IEC_Timer."TO_auf_CM05.QM64",
                  TO_schliessen := #IEC_Timer."TO_zu_CM05.QM64");
END_REGION

REGION Network 8 (SCL): GP01

   "Ventilstatus"(SRM_auf := "E_SRM_GP01.QM14_auf",
                  SRM_zu := "E_SRM_GP01.QM14_zu",
                  A_Ventil := "A_GP01.QM14",
                  Zeit := #Param.TO,
                  "Farbe HMI" => "Panel".Ventil."GP01.QM14",
                  Mld_Sensorfehler := #Mld."SF_GP01.QM14",
                  Mld_TO_oeffnen => #Mld."TO_auf_GP01.QM14",
                  Mld_TO_schliessen => #Mld."TO_zu_GP01.QM14",
                  TO_oeffnen := #IEC_Timer."TO_auf_GP01.QM14",
                  TO_schliessen := #IEC_Timer."TO_zu_GP01.QM14");

   "Ventilstatus"(SRM_auf := "E_SRM_GP01.QM15_auf",
                  SRM_zu := "E_SRM_GP01.QM15_zu",
                  A_Ventil := "A_GP01.QM15",
                  Zeit := #Param.TO,
                  "Farbe HMI" => "Panel".Ventil."GP01.QM15",
                  Mld_Sensorfehler := #Mld."SF_GP01.QM15",
                  Mld_TO_oeffnen => #Mld."TO_auf_GP01.QM15",
                  Mld_TO_schliessen => #Mld."TO_zu_GP01.QM15",
                  TO_oeffnen := #IEC_Timer."TO_auf_GP01.QM15",
                  TO_schliessen := #IEC_Timer."TO_zu_GP01.QM15");

   "Ventilstatus"(SRM_auf := "E_SRM_GP01.QM16_auf",
                  SRM_zu := "E_SRM_GP01.QM16_zu",
                  A_Ventil := "A_GP01.QM16",
                  Zeit := #Param.TO,
                  "Farbe HMI" => "Panel".Ventil."GP01.QM16",
                  Mld_Sensorfehler := #Mld."SF_GP01.QM16",
                  Mld_TO_oeffnen => #Mld."TO_auf_GP01.QM16",
                  Mld_TO_schliessen => #Mld."TO_zu_GP01.QM16",
                  TO_oeffnen := #IEC_Timer."TO_auf_GP01.QM16",
                  TO_schliessen := #IEC_Timer."TO_zu_GP01.QM16");

   "Ventilstatus"(SRM_auf := "E_SRM_GP01.QM17_auf",
                  SRM_zu := "E_SRM_GP01.QM17_zu",
                  A_Ventil := "A_GP01.QM17",
                  Zeit := #Param.TO,
                  "Farbe HMI" => "Panel".Ventil."GP01.QM17",
                  Mld_Sensorfehler := #Mld."SF_GP01.QM17",
                  Mld_TO_oeffnen => #Mld."TO_auf_GP01.QM17",
                  Mld_TO_schliessen => #Mld."TO_zu_GP01.QM17",
                  TO_oeffnen := #IEC_Timer."TO_auf_GP01.QM17",
                  TO_schliessen := #IEC_Timer."TO_zu_GP01.QM17");

   "Ventilstatus"(SRM_auf := "E_SRM_GP01.QM18_auf",
                  SRM_zu := "E_SRM_GP01.QM18_zu",
                  A_Ventil := "A_GP01.QM18",
                  Zeit := #Param.TO,
                  "Farbe HMI" => "Panel".Ventil."GP01.QM18",
                  Mld_Sensorfehler := #Mld."SF_GP01.QM18",
                  Mld_TO_oeffnen => #Mld."TO_auf_GP01.QM18",
                  Mld_TO_schliessen => #Mld."TO_zu_GP01.QM18",
                  TO_oeffnen := #IEC_Timer."TO_auf_GP01.QM18",
                  TO_schliessen := #IEC_Timer."TO_zu_GP01.QM18");

   "Ventilstatus"(SRM_auf := "E_SRM_GP01.QM19_auf",
                  SRM_zu := "E_SRM_GP01.QM19_zu",
                  A_Ventil := "A_GP01.QM19",
                  Zeit := #Param.TO,
                  "Farbe HMI" => "Panel".Ventil."GP01.QM19",
                  Mld_Sensorfehler := #Mld."SF_GP01.QM19",
                  Mld_TO_oeffnen => #Mld."TO_auf_GP01.QM19",
                  Mld_TO_schliessen => #Mld."TO_zu_GP01.QM19",
                  TO_oeffnen := #IEC_Timer."TO_auf_GP01.QM19",
                  TO_schliessen := #IEC_Timer."TO_zu_GP01.QM19");

   "Ventilstatus"(SRM_auf := "E_SRM_GP01.QM20_auf",
                  SRM_zu := "E_SRM_GP01.QM20_zu",
                  A_Ventil := "A_GP01.QM20",
                  Zeit := #Param.TO,
                  "Farbe HMI" => "Panel".Ventil."GP01.QM20",
                  Mld_Sensorfehler := #Mld."SF_GP01.QM20",
                  Mld_TO_oeffnen => #Mld."TO_auf_GP01.QM20",
                  Mld_TO_schliessen => #Mld."TO_zu_GP01.QM20",
                  TO_oeffnen := #IEC_Timer."TO_auf_GP01.QM20",
                  TO_schliessen := #IEC_Timer."TO_zu_GP01.QM20");

   "Ventilstatus"(SRM_auf := "E_SRM_GP01.QM21_auf",
                  SRM_zu := "E_SRM_GP01.QM21_zu",
                  A_Ventil := "A_GP01.QM21",
                  Zeit := #Param.TO,
                  "Farbe HMI" => "Panel".Ventil."GP01.QM21",
                  Mld_Sensorfehler := #Mld."SF_GP01.QM21",
                  Mld_TO_oeffnen => #Mld."TO_auf_GP01.QM21",
                  Mld_TO_schliessen => #Mld."TO_zu_GP01.QM21",
                  TO_oeffnen := #IEC_Timer."TO_auf_GP01.QM21",
                  TO_schliessen := #IEC_Timer."TO_zu_GP01.QM21");

   "Ventilstatus"(SRM_auf := "E_SRM_GP01.QM22_auf",
                  SRM_zu := "E_SRM_GP01.QM22_zu",
                  A_Ventil := "A_GP01.QM22",
                  Zeit := #Param.TO,
                  "Farbe HMI" => "Panel".Ventil."GP01.QM22",
                  Mld_Sensorfehler := #Mld."SF_GP01.QM22",
                  Mld_TO_oeffnen => #Mld."TO_auf_GP01.QM22",
                  Mld_TO_schliessen => #Mld."TO_zu_GP01.QM22",
                  TO_oeffnen := #IEC_Timer."TO_auf_GP01.QM22",
                  TO_schliessen := #IEC_Timer."TO_zu_GP01.QM22");

   "Ventilstatus_einfach"(A_Ventil:="A_GP01.QM23",
                          "Farbe HMI"=> "Panel".Ventil."GP01.QM23");
END_REGION

REGION Network 9 (SCL): GP02
   "Ventilstatus_einfach"(A_Ventil := "A_GP02.QM37",
                          "Farbe HMI" => "Panel".Ventil."GP02.QM37");

   "Ventilstatus"(SRM_auf := "E_SRM_GP02.QM38_auf",
                  SRM_zu := "E_SRM_GP02.QM38_zu",
                  A_Ventil := "A_GP02.QM38",
                  Zeit := #Param.TO,
                  "Farbe HMI" => "Panel".Ventil."GP02.QM38",
                  Mld_Sensorfehler := #Mld."SF_GP02.QM38",
                  Mld_TO_oeffnen => #Mld."TO_auf_GP02.QM38",
                  Mld_TO_schliessen => #Mld."TO_zu_GP02.QM38",
                  TO_oeffnen := #IEC_Timer."TO_auf_GP02.QM38",
                  TO_schliessen := #IEC_Timer."TO_zu_GP02.QM38");

   "Ventilstatus"(SRM_auf := "E_SRM_GP02.QM39_auf",
                  SRM_zu := "E_SRM_GP02.QM39_zu",
                  A_Ventil := "A_GP02.QM39",
                  Zeit := #Param.TO,
                  "Farbe HMI" => "Panel".Ventil."GP02.QM39",
                  Mld_Sensorfehler := #Mld."SF_GP02.QM39",
                  Mld_TO_oeffnen => #Mld."TO_auf_GP02.QM39",
                  Mld_TO_schliessen => #Mld."TO_zu_GP02.QM39",
                  TO_oeffnen := #IEC_Timer."TO_auf_GP02.QM39",
                  TO_schliessen := #IEC_Timer."TO_zu_GP02.QM39");

   "Ventilstatus"(SRM_auf := "E_SRM_GP02.QM40_auf",
                  SRM_zu := "E_SRM_GP02.QM40_zu",
                  A_Ventil := "A_GP02.QM40",
                  Zeit := #Param.TO,
                  "Farbe HMI" => "Panel".Ventil."GP02.QM40",
                  Mld_Sensorfehler := #Mld."SF_GP02.QM40",
                  Mld_TO_oeffnen => #Mld."TO_auf_GP02.QM40",
                  Mld_TO_schliessen => #Mld."TO_zu_GP02.QM40",
                  TO_oeffnen := #IEC_Timer."TO_auf_GP02.QM40",
                  TO_schliessen := #IEC_Timer."TO_zu_GP02.QM40");

   "Ventilstatus"(SRM_auf := "E_SRM_GP02.QM41_auf",
                  SRM_zu := "E_SRM_GP02.QM41_zu",
                  A_Ventil := "A_GP02.QM41",
                  Zeit := #Param.TO,
                  "Farbe HMI" => "Panel".Ventil."GP02.QM41",
                  Mld_Sensorfehler := #Mld."SF_GP02.QM41",
                  Mld_TO_oeffnen => #Mld."TO_auf_GP02.QM41",
                  Mld_TO_schliessen => #Mld."TO_zu_GP02.QM41",
                  TO_oeffnen := #IEC_Timer."TO_auf_GP02.QM41",
                  TO_schliessen := #IEC_Timer."TO_zu_GP02.QM41");

   "Ventilstatus"(SRM_auf := "E_SRM_GP02.QM42_auf",
                  SRM_zu := "E_SRM_GP02.QM42_zu",
                  A_Ventil := "A_GP02.QM42",
                  Zeit := #Param.TO,
                  "Farbe HMI" => "Panel".Ventil."GP02.QM42",
                  Mld_Sensorfehler := #Mld."SF_GP02.QM42",
                  Mld_TO_oeffnen => #Mld."TO_auf_GP02.QM42",
                  Mld_TO_schliessen => #Mld."TO_zu_GP02.QM41",
                  TO_oeffnen := #IEC_Timer."TO_auf_GP02.QM42",
                  TO_schliessen := #IEC_Timer."TO_zu_GP02.QM42");

   "Ventilstatus"(SRM_auf := "DB_PNOZ_IN_Out".In."SRM_Auf_BG-QM43",
                  SRM_zu := "DB_PNOZ_IN_Out".In."SRM_Zu_BG-QM43",
                  A_Ventil := "A_GP02.QM43",
                  Zeit := #Param.TO,
                  "Farbe HMI" => "Panel".Ventil."GP02.QM43",
                  Mld_Sensorfehler := #Mld."SF_GP02.QM43",
                  Mld_TO_oeffnen => #Mld."TO_auf_GP02.QM43",
                  Mld_TO_schliessen => #Mld."TO_zu_GP02.QM43",
                  TO_oeffnen := #IEC_Timer."TO_auf_GP02.QM43",
                  TO_schliessen := #IEC_Timer."TO_zu_GP02.QM43");

   "Ventilstatus"(SRM_auf := "DB_PNOZ_IN_Out".In."SRM_Auf_BG-QM44",
                  SRM_zu := "DB_PNOZ_IN_Out".In."SRM_Zu_BG-QM44",
                  A_Ventil := "A_GP02.QM44",
                  Zeit := #Param.TO,
                  "Farbe HMI" => "Panel".Ventil."GP02.QM44",
                  Mld_Sensorfehler := #Mld."SF_GP02.QM44",
                  Mld_TO_oeffnen => #Mld."TO_auf_GP02.QM44",
                  Mld_TO_schliessen => #Mld."TO_zu_GP02.QM44",
                  TO_oeffnen := #IEC_Timer."TO_auf_GP02.QM44",
                  TO_schliessen := #IEC_Timer."TO_zu_GP02.QM44");

   "Ventilstatus"(SRM_auf := "E_SRM_GP02.QM45_auf",
                  SRM_zu := "E_SRM_GP02.QM45_zu",
                  A_Ventil := "A_GP02.QM45",
                  Zeit := #Param.TO,
                  "Farbe HMI" => "Panel".Ventil."GP02.QM45",
                  Mld_Sensorfehler := #Mld."SF_GP02.QM45",
                  Mld_TO_oeffnen => #Mld."TO_auf_GP02.QM45",
                  Mld_TO_schliessen => #Mld."TO_zu_GP02.QM45",
                  TO_oeffnen := #IEC_Timer."TO_auf_GP02.QM45",
                  TO_schliessen := #IEC_Timer."TO_zu_GP02.QM45");

   "Ventilstatus"(SRM_auf := "E_SRM_GP02.QM46_auf",
                  SRM_zu := "E_SRM_GP02.QM46_zu",
                  A_Ventil := "A_GP02.QM46",
                  Zeit := #Param.TO,
                  "Farbe HMI" => "Panel".Ventil."GP02.QM46",
                  Mld_Sensorfehler := #Mld."SF_GP02.QM46",
                  Mld_TO_oeffnen => #Mld."TO_auf_GP02.QM46",
                  Mld_TO_schliessen => #Mld."TO_zu_GP02.QM46",
                  TO_oeffnen := #IEC_Timer."TO_auf_GP02.QM46",
                  TO_schliessen := #IEC_Timer."TO_zu_GP02.QM46");
END_REGION

REGION Network 10 (SCL): CL0x
   "Ventilstatus_einfach"(A_Ventil:= "A_CL01.QM51",
                          "Farbe HMI" => "Panel".Ventil."CL01.QM51");

   "Ventilstatus_einfach"(A_Ventil := "A_CL02.QM52",
                          "Farbe HMI" => "Panel".Ventil."CL02.QM52");
END_REGION
END_FUNCTION_BLOCK

FUNCTION "FC_Niveau_St" : Void   // FC96, STL
TITLE = Badniveau-Steuerungen
{ S7_Optimized_Access := 'FALSE' }
AUTHOR : RE
NAME : FC_nass
VERSION : 2.0
// stored: AutoNumber false
   VAR_TEMP
      Freigabe : Bool;
   END_VAR
BEGIN

NETWORK
TITLE = Niveau-Regelungen/Nachspeisungen/Spritzregister
      CLR;
      =     "DB_NSP".Test_on;

      CALL  "FC_Nachspeisung";

      A     "DB_ANLAGE".BA.Simulation;
      BEC;


NETWORK
TITLE = CM01
      A     "Panel".CM01.NSP_Auto;
      =     "DB_Panel_Posinfo".Pos[1].NS_Auto;

// Becken leer und keine Dosierung aktiv
      AN    "DB_POS".POS[1].belegt;
      AN    "DB_POS".POS[2].belegt;
      AN    "DB_POS".POS[3].belegt;
      AN    "DB_POS".POS[4].belegt;
      AN    "DB_POS".POS[5].belegt;
      AN    "DB_POS".POS[6].belegt;
      AN    "DB_DP".DP[1].Dosi_akt;
      AN    "DB_DP".DP[2].Dosi_akt;
      AN    "DB_DP".DP[5].Dosi_akt;
      AN    "DB_DP".DP[6].Dosi_akt;
      =     "DB_NSP".NSP[1].Freigabe;

      A     "E_Niv_Min_CM01.BL03";
      =     "DB_NSP".NSP[1].Niveau_ok;
      =     "DB_NSP".NSP[2].Niveau_ok;
      =     "DB_NSP".NSP[3].Niveau_ok;
      =     "DB_NSP".NSP[4].Niveau_ok;
      =     "DB_NSP".NSP[5].Niveau_ok;
      =     "DB_NSP".NSP[6].Niveau_ok;
      NOT;
      =     "DB_NSP".NSP[1].AL_Niv_min;

// Dosierungen gegeneinander verriegeln
// Verwerfen hat Vorrang
      A     "DB_DP".DP[1].Dosi_akt;
      O     "DB_DP".DP[5].Dosi_akt;
      O     "DB_DP".DP[3].Dosi_akt;
      O     "DB_DP".DP[7].Dosi_akt;
      S     "DB_DP".DP[2].DP_OFF;
      S     "DB_DP".DP[6].DP_OFF;
      S     "DB_DP".DP[4].DP_OFF;
      S     "DB_DP".DP[8].DP_OFF;
      JC    Ents;

// CM01 gewinnt
      A     "DB_DP".DP[2].Dosi_akt;  //CM01
      O     "DB_DP".DP[6].Dosi_akt;
      A(;
      A     "DB_DP".DP[4].Dosi_akt;  //CM02
      O     "DB_DP".DP[8].Dosi_akt;
      );
      AN    "DB_DP".DP[2].DP_OFF;
      AN    "DB_DP".DP[6].DP_OFF;
      S     "DB_DP".DP[4].DP_OFF;
      S     "DB_DP".DP[8].DP_OFF;
      JC    Ents;

      A     "DB_DP".DP[2].Dosi_akt;  //CM01
      O     "DB_DP".DP[6].Dosi_akt;
      AN    "DB_DP".DP[2].DP_OFF;
      AN    "DB_DP".DP[6].DP_OFF;
      =     "DB_DP".DP[4].DP_OFF;
      =     "DB_DP".DP[8].DP_OFF;

      A     "DB_DP".DP[4].Dosi_akt;  //CM02
      O     "DB_DP".DP[8].Dosi_akt;
      AN    "DB_DP".DP[4].DP_OFF;
      AN    "DB_DP".DP[8].DP_OFF;
      =     "DB_DP".DP[2].DP_OFF;
      =     "DB_DP".DP[6].DP_OFF;

//Verwerfen - alles aus
Ents: AN    "DB_DP".DP[1].Dosi_akt;
      AN    "DB_DP".DP[3].Dosi_akt;
      AN    "DB_DP".DP[5].Dosi_akt;
      AN    "DB_DP".DP[7].Dosi_akt;
      R     "DB_DP".DP[1].DP_OFF;
      R     "DB_DP".DP[3].DP_OFF;
      R     "DB_DP".DP[5].DP_OFF;
      R     "DB_DP".DP[7].DP_OFF;

// Verwerfen CM01 gewinnt
      A     "DB_DP".DP[1].Dosi_akt;  //CM01
      O     "DB_DP".DP[5].Dosi_akt;
      A(;
      A     "DB_DP".DP[3].Dosi_akt;  //CM02
      O     "DB_DP".DP[7].Dosi_akt;
      );
      AN    "DB_DP".DP[1].DP_OFF;
      AN    "DB_DP".DP[5].DP_OFF;
      S     "DB_DP".DP[3].DP_OFF;
      S     "DB_DP".DP[7].DP_OFF;
      JC    CM01;

      A     "DB_DP".DP[1].Dosi_akt;  //CM01
      O     "DB_DP".DP[5].Dosi_akt;
      AN    "DB_DP".DP[1].DP_OFF;
      AN    "DB_DP".DP[5].DP_OFF;
      =     "DB_DP".DP[3].DP_OFF;
      =     "DB_DP".DP[7].DP_OFF;

      A     "DB_DP".DP[3].Dosi_akt;  //CM02
      O     "DB_DP".DP[7].Dosi_akt;
      AN    "DB_DP".DP[3].DP_OFF;
      AN    "DB_DP".DP[7].DP_OFF;
      =     "DB_DP".DP[1].DP_OFF;
      =     "DB_DP".DP[5].DP_OFF;

CM01: NOP   0;
// Anforderung bilden
// Nachschärfen
      A     "DB_NSP".NSP[1].Nachspeisen;
      O(;
      A     "DB_DP".DP[2].Dosi_akt;
      AN    "DB_DP".DP[2].DP_OFF;
      );
      O(;
      A     "DB_DP".DP[6].Dosi_akt;
      AN    "DB_DP".DP[6].DP_OFF;
      );
      A     "Pu_GP01.GP13".In.Auto;
      A     "Pu_GP01.GP13".Out.Versorgung_UV01;
      AN    "Pu_GP02.GP10".In.Anf_HF_CM01;
      =     "Pu_GP01.GP13".In.Anf_HF_CM01;

      A     "DB_NSP".NSP[1].Nachspeisen;
      O(;
      A     "DB_DP".DP[2].Dosi_akt;
      AN    "DB_DP".DP[2].DP_OFF;
      );
      O(;
      A     "DB_DP".DP[6].Dosi_akt;
      AN    "DB_DP".DP[6].DP_OFF;
      );
      A     "Pu_GP02.GP10".In.Auto;
      A     "Pu_GP02.GP10".Out.Versorgung_UV01;
      AN    "Pu_GP01.GP13".In.Anf_HF_CM01;
      =     "Pu_GP02.GP10".In.Anf_HF_CM01;

// Verwerfen
      A     "DB_DP".DP[1].Dosi_akt;
      AN    "DB_DP".DP[1].DP_OFF;
      O(;
      A     "DB_DP".DP[5].Dosi_akt;
      AN    "DB_DP".DP[5].DP_OFF;
      );
      A     "UP_CM01.GP02".In.Auto;
      A(;
      A     "UP_CM01.GP02".In."SRM_GP01.QM14_auf";
      O     "UP_CM01.GP02".In."SRM_GP02.QM41_auf";
      );
      =     "UP_CM01.GP02".In.Anf_HF_Ents_CM0x;

// WT-zählergesteuert (DP1/2)
      A     "Panel".CM01.Dosierung_LF;
      R     "DB_Panel_DP".DoPu[1].Auto;
      R     "DB_Panel_DP".DoPu[2].Auto;

// LF-gesteuert (DP(5/6)
      CALL  "ToDo";

      A     "DB_DP".DP[5].Dosi_akt;
      O     "DB_DP".DP[6].Dosi_akt;
      L     S5T#15m;
      SF    "TA-Pause_LF_CM01";

      AN    "Panel".CM01.Dosierung_LF;
      R     "DB_Panel_DP".DoPu[5].Auto;
      R     "DB_Panel_DP".DoPu[6].Auto;
      JC    LF1E;

      L     "Panel".IW."LF_CM01.BN02";
      L     "Panel".CM01.Sollwert_LF;
      <R;  // ???
      AN    "TA-Pause_LF_CM01";
      AN    "DB_DP".DP[5].AM_DP_Start;
      AN    "DB_DP".DP[6].AM_DP_Start;
      S     "DB_DP".DP[5].DP_Start;
      S     "DB_DP".DP[5].AM_DP_Start;
      S     "DB_DP".DP[6].DP_Start;
      S     "DB_DP".DP[6].AM_DP_Start;
      JC    LF1E;

      A     "DB_DP".DP[5].Dosi_akt;
      R     "DB_DP".DP[5].AM_DP_Start;

      A     "DB_DP".DP[6].Dosi_akt;
      R     "DB_DP".DP[6].AM_DP_Start;

LF1E: NOP   0;


NETWORK
TITLE = CM02
      A     "Panel".CM02.NSP_Auto;
      =     "DB_Panel_Posinfo".Pos[13].NS_Auto;

// Becken leer und keine Dosierung aktiv
      AN    "DB_POS".POS[13].belegt;
      AN    "DB_POS".POS[14].belegt;
      AN    "DB_POS".POS[15].belegt;
      AN    "DB_POS".POS[16].belegt;
      AN    "DB_POS".POS[17].belegt;
      AN    "DB_POS".POS[18].belegt;
      AN    "DB_DP".DP[3].Dosi_akt;
      AN    "DB_DP".DP[4].Dosi_akt;
      AN    "DB_DP".DP[7].Dosi_akt;
      AN    "DB_DP".DP[8].Dosi_akt;
      =     "DB_NSP".NSP[13].Freigabe;

      A     "E_Niv_Min_CM02.BL10";
      =     "DB_NSP".NSP[13].Niveau_ok;
      =     "DB_NSP".NSP[14].Niveau_ok;
      =     "DB_NSP".NSP[15].Niveau_ok;
      =     "DB_NSP".NSP[16].Niveau_ok;
      =     "DB_NSP".NSP[17].Niveau_ok;
      =     "DB_NSP".NSP[18].Niveau_ok;
      NOT;
      =     "DB_NSP".NSP[13].AL_Niv_min;


// Anforderung bilden
// Nachschärfen
      A     "DB_NSP".NSP[13].Nachspeisen;
      O(;
      A     "DB_DP".DP[4].Dosi_akt;
      AN    "DB_DP".DP[4].DP_OFF;
      );
      O(;
      A     "DB_DP".DP[8].Dosi_akt;
      AN    "DB_DP".DP[8].DP_OFF;
      );
      A     "Pu_GP01.GP13".In.Auto;
      A     "Pu_GP01.GP13".Out.Versorgung_UV01;
      AN    "Pu_GP02.GP10".In.Anf_HF_CM02;
      =     "Pu_GP01.GP13".In.Anf_HF_CM02;

      A     "DB_NSP".NSP[13].Nachspeisen;
      O(;
      A     "DB_DP".DP[4].Dosi_akt;
      AN    "DB_DP".DP[4].DP_OFF;
      );
      O(;
      A     "DB_DP".DP[8].Dosi_akt;
      AN    "DB_DP".DP[8].DP_OFF;
      );
      A     "Pu_GP02.GP10".In.Auto;
      A     "Pu_GP02.GP10".Out.Versorgung_UV01;
      AN    "Pu_GP01.GP13".In.Anf_HF_CM02;
      =     "Pu_GP02.GP10".In.Anf_HF_CM02;

// Verwerfen
      A     "DB_DP".DP[3].Dosi_akt;
      AN    "DB_DP".DP[3].DP_OFF;
      O(;
      A     "DB_DP".DP[7].Dosi_akt;
      AN    "DB_DP".DP[7].DP_OFF;
      );
      A     "UP_CM02.GP05".In.Auto;
      A(;
      A     "UP_CM02.GP05".In."SRM_GP01.QM14_auf";
      O     "UP_CM02.GP05".In."SRM_GP02.QM41_auf";
      );
      =     "UP_CM02.GP05".In.Anf_HF_Ents_CM0x;

// WT-zählergesteuert (DP3/4)
      A     "Panel".CM02.Dosierung_LF;
      R     "DB_Panel_DP".DoPu[3].Auto;
      R     "DB_Panel_DP".DoPu[4].Auto;

// LF-gesteuert (DP(7/8)
      CALL  "ToDo";

      A     "DB_DP".DP[7].Dosi_akt;
      O     "DB_DP".DP[8].Dosi_akt;
      L     S5T#15m;
      SF    "TA-Pause_LF_CM02";

      AN    "Panel".CM02.Dosierung_LF;
      R     "DB_Panel_DP".DoPu[7].Auto;
      R     "DB_Panel_DP".DoPu[8].Auto;
      JC    LF2E;

      L     "Panel".IW."LF_CM02.BN04";
      L     "Panel".CM02.Sollwert_LF;
      <R;  // ???
      AN    "TA-Pause_LF_CM02";
      AN    "DB_DP".DP[7].AM_DP_Start;
      AN    "DB_DP".DP[8].AM_DP_Start;
      S     "DB_DP".DP[7].DP_Start;
      S     "DB_DP".DP[7].AM_DP_Start;
      S     "DB_DP".DP[8].DP_Start;
      S     "DB_DP".DP[8].AM_DP_Start;
      JC    LF2E;

      A     "DB_DP".DP[7].Dosi_akt;
      R     "DB_DP".DP[7].AM_DP_Start;

      A     "DB_DP".DP[8].Dosi_akt;
      R     "DB_DP".DP[8].AM_DP_Start;

LF2E: NOP   0;


NETWORK
TITLE = CM03

      A     "Panel".CM03.SPR_Auto;
      =     "DB_Panel_Posinfo".Pos[7].SR_Auto;
      =     "DB_Panel_Posinfo".Pos[8].SR_Auto;
      =     "DB_Panel_Posinfo".Pos[9].SR_Auto;
      =     "DB_Panel_Posinfo".Pos[10].SR_Auto;
      =     "DB_Panel_Posinfo".Pos[11].SR_Auto;
      =     "DB_Panel_Posinfo".Pos[12].SR_Auto;

      A     "Panel".CM03.SPR_Start_Test;
      R     "Panel".CM03.SPR_Start_Test;
      JCN   ST03;
      L     "Panel".CM03.SPR_Zeit_Test;
      T     "DB_Panel_Posinfo".Pos[7].T_Zt_SR;

ST03: A     "Panel".CM03.SPR_Stopp_Test;
      R     "Panel".CM03.SPR_Stopp_Test;
      JCN   FN03;
      L     0;
      T     "DB_Panel_Posinfo".Pos[7].T_Zt_SR;

//Pos.7..12
FN03: AN    "T_VEW_niO";
      A     "E_Niv_Uel_CM05.BL12";
      =     "DB_NSP".NSP[7].Freigabe;
      =     "DB_NSP".NSP[8].Freigabe;
      =     "DB_NSP".NSP[9].Freigabe;
      =     "DB_NSP".NSP[10].Freigabe;
      =     "DB_NSP".NSP[11].Freigabe;
      =     "DB_NSP".NSP[12].Freigabe;

// Spritzregister: beim Heben und Senken
      A     "DB_NSP".NSP[7].Spritzen;
      O     "DB_NSP".NSP[8].Spritzen;
      O     "DB_NSP".NSP[9].Spritzen;
      O     "DB_NSP".NSP[10].Spritzen;
      O     "DB_NSP".NSP[11].Spritzen;
      O     "DB_NSP".NSP[12].Spritzen;
      AN    "T_VEW_niO";
      A     "E_Niv_Uel_CM05.BL12";
      =     "A_CM03.QM35";


NETWORK
TITLE = CM04
//Pos.19..24
      A     "Panel".CM04.SPR_Auto;
      =     "DB_Panel_Posinfo".Pos[19].SR_Auto;
      =     "DB_Panel_Posinfo".Pos[20].SR_Auto;
      =     "DB_Panel_Posinfo".Pos[21].SR_Auto;
      =     "DB_Panel_Posinfo".Pos[22].SR_Auto;
      =     "DB_Panel_Posinfo".Pos[23].SR_Auto;
      =     "DB_Panel_Posinfo".Pos[24].SR_Auto;

      A     "Panel".CM04.NSP_Auto;
      =     "DB_Panel_Posinfo".Pos[19].NS_Auto;
      =     "DB_Panel_Posinfo".Pos[20].NS_Auto;
      =     "DB_Panel_Posinfo".Pos[21].NS_Auto;
      =     "DB_Panel_Posinfo".Pos[22].NS_Auto;
      =     "DB_Panel_Posinfo".Pos[23].NS_Auto;
      =     "DB_Panel_Posinfo".Pos[24].NS_Auto;

      L     "Panel".CM04.NSP_Zeit;
      T     "DB_Panel_Posinfo".Pos[19].Zeit_NS;
      T     "DB_Panel_Posinfo".Pos[20].Zeit_NS;
      T     "DB_Panel_Posinfo".Pos[21].Zeit_NS;
      T     "DB_Panel_Posinfo".Pos[22].Zeit_NS;
      T     "DB_Panel_Posinfo".Pos[23].Zeit_NS;
      T     "DB_Panel_Posinfo".Pos[24].Zeit_NS;

      A     "Panel".CM04.SPR_Start_Test;
      R     "Panel".CM04.SPR_Start_Test;
      JCN   ST04;
      L     "Panel".CM04.SPR_Zeit_Test;
      T     "DB_Panel_Posinfo".Pos[19].T_Zt_SR;

ST04: A     "Panel".CM04.SPR_Stopp_Test;
      R     "Panel".CM04.SPR_Stopp_Test;
      JCN   NS04;
      L     0;
      T     "DB_Panel_Posinfo".Pos[19].T_Zt_SR;

NS04: A     "Panel".CM04.NSP_Start_Test;
      R     "Panel".CM04.NSP_Start_Test;
      JCN   SN04;
      L     "Panel".CM04.NSP_Zeit_Tes;
      T     "DB_Panel_Posinfo".Pos[19].T_Zt_NS;

SN04: A     "Panel".CM04.NSP_Stopp_Test;
      R     "Panel".CM04.NSP_Stopp_Test;
      JCN   FN04;
      L     0;
      T     "DB_Panel_Posinfo".Pos[19].T_Zt_NS;

FN04: AN    "T_VEW_niO";
      A     "E_Niv_Uel_CM05.BL12";
      =     "DB_NSP".NSP[19].Freigabe;
      =     "DB_NSP".NSP[20].Freigabe;
      =     "DB_NSP".NSP[21].Freigabe;
      =     "DB_NSP".NSP[22].Freigabe;
      =     "DB_NSP".NSP[23].Freigabe;
      =     "DB_NSP".NSP[24].Freigabe;

// Spritzregister: beim Heben
      A     "DB_NSP".NSP[19].Spritzen;
      O     "DB_NSP".NSP[20].Spritzen;
      O     "DB_NSP".NSP[21].Spritzen;
      O     "DB_NSP".NSP[22].Spritzen;
      O     "DB_NSP".NSP[23].Spritzen;
      O     "DB_NSP".NSP[24].Spritzen;
      AN    "T_VEW_niO";
      A     "E_Niv_Uel_CM05.BL12";
      =     "A_CM04.QM74";

// Nachspeisung
// Zeit pro Korb
// niveaugesteuert, wenn CM03 nicht belegt und "min"-Niveau nicht erreicht

      A     "E_Niv_Min_CM03.BL06";
      O     "DB_POS".POS[7].belegt;
      O     "DB_POS".POS[8].belegt;
      O     "DB_POS".POS[9].belegt;
      O     "DB_POS".POS[10].belegt;
      O     "DB_POS".POS[11].belegt;
      O     "DB_POS".POS[12].belegt;
      O     "A_CM04.QM74";
      =     "DB_NSP".NSP[19].Niveau_ok;
      =     "DB_NSP".NSP[20].Niveau_ok;
      =     "DB_NSP".NSP[21].Niveau_ok;
      =     "DB_NSP".NSP[22].Niveau_ok;
      =     "DB_NSP".NSP[23].Niveau_ok;
      =     "DB_NSP".NSP[24].Niveau_ok;
      NOT;  // Nicht Spritzen und Nachspeisen gleichzeitig
      =     "DB_NSP".NSP[19].AL_Niv_min;

// Nicht Spritzen und Nachspeisen gleichzeitig
      A     "DB_POS".POS[19].FW_Hebt;
      =     "DB_NSP".NSP[19].Warte_NSPT;
      A     "DB_POS".POS[20].FW_Hebt;
      =     "DB_NSP".NSP[20].Warte_NSPT;
      A     "DB_POS".POS[21].FW_Hebt;
      =     "DB_NSP".NSP[21].Warte_NSPT;
      A     "DB_POS".POS[22].FW_Hebt;
      =     "DB_NSP".NSP[22].Warte_NSPT;
      A     "DB_POS".POS[23].FW_Hebt;
      =     "DB_NSP".NSP[23].Warte_NSPT;
      A     "DB_POS".POS[24].FW_Hebt;
      =     "DB_NSP".NSP[24].Warte_NSPT;

      A     "DB_NSP".NSP[19].Nachspeisen;
      O     "DB_NSP".NSP[20].Nachspeisen;
      O     "DB_NSP".NSP[21].Nachspeisen;
      O     "DB_NSP".NSP[22].Nachspeisen;
      O     "DB_NSP".NSP[23].Nachspeisen;
      O     "DB_NSP".NSP[24].Nachspeisen;
      =     "A_CM04.QM77";

END_FUNCTION

FUNCTION "FC_Nachspeisung" : Void   // FC97, STL
TITLE = Nachspeisung
{ S7_Optimized_Access := 'FALSE' }
// stored: AutoNumber false
   VAR_TEMP
      Adr_NSP_DB : DWord;
      Adr_PosInfo_DB : DWord;
      Adr_Overview_DB : DWord;
      Adr_Pos_DB : DWord;
      FW_DI_Nr : Word;
      Count : Int;
      Restzeit_NS : Int;
      Restzeit_SPR : Int;
      TestZeit_NS : Int;
      TestZeit_SPR : Int;
      Zeit_NS : Int;
      Zeit_SPR : Int;
      NS_Kor_Tr : Byte;
      Coun_Kor : Byte;
      Pos_Nr : Byte;
      AL_Nr : USInt;
      FW_Nr : Byte;
      Akt_Hub_Inc : Byte;
      NSP_erlaubt : Bool;
      NS_Niv : Bool;
      NST_in : Bool;
      NST_out : Bool;
      Trommel : Bool;
      Freigabe : Bool;
      ext_Start : Bool;
      Niveau_ok : Bool;
      belegt : Bool;
      Leer_WT : Bool;
      Hebt : Bool;
      Senkt : Bool;
      Bearbeitung : Bool;
      Eingesetzt : Bool;
      Ausgehoben : Bool;
      AM_Belegt : Bool;
      AM_min : Bool;
      AM_AL_Zeit : Bool;
      AL_Uel : Bool;
      AL_min : Bool;
      AL_Zeit : Bool;
      AL_Send : Bool;
      neu : Bool;
      SPR_free : Bool;
      NSP_free : Bool;
      NS_akt : Bool;
      SPR_on : Bool;
      SPR_out : Bool;
      SPR_in : Bool;
      SPR_exp : Bool;
      SPR_Zeit : Bool;
      SPR_erlaubt : Bool;
      Simu : Bool;
      AM_Uel : Bool;
      Reset : Bool;
      evt : Bool;
      AL_NS : Bool;
      hupen : Bool;
      NS_On : Bool;
      SPR_off : Bool;
      Spr_frg : Bool;
      Wait_NSPT : Bool;
   END_VAR
BEGIN

NETWORK
TITLE = AMS-Reset
      A     "DB_ANLAGE".IN.AMS_Restart;
      S     "DB_NSP".AMS_Reset;

      A     "DB_ANLAGE".IN.Quitt_Err;
      S     "DB_NSP".Reset;

NETWORK
TITLE = Schleife
      A     "Imp_1Hz";
      S     "DB_NSP".Sekunde;

      L     0;
      L     "DB_NSP".akt_NSP;
      <I;
      A(;
      L     "DB_ANLAGE".config.ANZ_Pos;
      <=I;
      );
      JC    ok;
      R     "DB_NSP".Test_akt;
      R     "DB_NSP".Test_start;

      L     1;
      T     "DB_NSP".akt_NSP;
      L     0;
      T     "DB_NSP".TestNr;

ok:   L     0;
      L     "DB_NSP".TestNr;
      ==I;
      R     "DB_NSP".Test_akt;

      A     "DB_NSP".Test_akt;
      R     "DB_NSP".Test_start;
      JC    pos;

      L     "DB_NSP".Anz_Per_Cyc;
ret:  T     #Count;

pos:  L     "DB_NSP".akt_NSP;
      T     #Pos_Nr;
      +     -1;
      L     "DB_NSP".leng;
      *D;
      L     "DB_NSP".Offset;
      +D;
      SLD   3;
      T     #Adr_NSP_DB;
      LAR1;
      OPNDI "DB_NSP";
      JU    Niv;

next: L     "DB_NSP".akt_NSP;
      L     "DB_ANLAGE".config.ANZ_Pos;
      <I;
      AN    "DB_NSP".Test_akt;
      JC    add;

      A     "DB_NSP".Sekunde;
      =     "DB_NSP".Takt;
      R     "DB_NSP".Sekunde;

      A     "DB_NSP".AMS_new;
      R     "DB_NSP".AMS_new;

      A     "DB_NSP".AMS_Reset;
      S     "DB_NSP".AMS_new;
      R     "DB_NSP".AMS_Reset;

      A     "DB_NSP".Test_akt;
      JC    end;

      A     "DB_NSP".Test_start;
      S     "DB_NSP".Test_akt;

      L     "DB_NSP".TestNr;
      A     "DB_NSP".Test_akt;
      JC    Test;

      A     "DB_NSP".temp_Warn;
      =     "DB_NSP".SammelWarn;
      R     "DB_NSP".temp_Warn;

      A     "DB_NSP".temp_STM;
      =     "DB_NSP".Sammelstoer;
      R     "DB_NSP".temp_STM;

      L     1;
Test: T     "DB_NSP".akt_NSP;

      L     0;
      L     "DB_NSP".TestNr;
      <>I;
      S     "DB_NSP".Test_start;
      JU    wtr;

add:  L     "DB_NSP".akt_NSP;
      +     1;
      T     "DB_NSP".akt_NSP;
wtr:  L     #Count;
      LOOP  ret;

end:  BE;

NETWORK
TITLE = Niveau regeln
Niv:  SET;
      R     #NS_On;
      R     #SPR_on;
      A     "DB_ANLAGE".BA.Simulation;
      =     #Simu;
      OPNDI "DB_NSP";
      A     DIX [AR1, P#2.0];  //Freigabe
      O     #Simu;
      =     #Freigabe;
      A     DIX [AR1, P#2.1];  //externer Start
      =     #ext_Start;
      A     DIX [AR1, P#2.2];  //Niveau ok
      =     #Niveau_ok;
      A     DIX [AR1, P#2.3];  //NS_akt
      =     #NS_akt;

      L     DIW [AR1, P#4.0];  //Restzeit
      T     #Restzeit_NS;
      L     DIW [AR1, P#8.0];  //Restzeit Spritzregister
      T     #Restzeit_SPR;

      L     DIW [AR1, P#12.0];  //"DB_NSP".NSP[1].RestVerz
      L     0;
      <=I;
      =     #AL_Send;

      L     DIW [AR1, P#16.0];  //"DB_NSP".NSP[1].RestNS_AL
      L     0;
      <=I;
      A(;
      L     DIW [AR1, P#14.0];  //"DB_NSP".NSP[1].VerzNS_AL
      <I;
      );
      =     #AL_NS;

      A     DIX [AR1, P#0.0];  //"DB_NSP".NSP[1].NSP
      =     #NS_Niv;
      A     DIX [AR1, P#0.1];  //"DB_NSP".NSP[1].NST_in
      =     #NST_in;
      A     DIX [AR1, P#0.2];  //"DB_NSP".NSP[1].NST_out
      =     #NST_out;
      A     DIX [AR1, P#0.3];  //"DB_NSP".NSP[1].SPR_in
      =     #SPR_in;
      A     DIX [AR1, P#0.4];  //"DB_NSP".NSP[1].SPR_out
      =     #SPR_out;
      A     DIX [AR1, P#0.5];  //"DB_NSP".NSP[1].SPR_expo
      =     #SPR_exp;
      A     DIX [AR1, P#0.6];  //"DB_NSP".NSP[1].SPR_Zeit
      =     #SPR_Zeit;
      A     DIX [AR1, P#18.0];  //"DB_NSP".NSP[1].AM_AL_min
      =     #AM_min;
      A     DIX [AR1, P#18.1];  //"DB_NSP".NSP[1].AM_AL_Uel
      =     #AM_Uel;
      A     DIX [AR1, P#18.2];  //"DB_NSP".NSP[1].AM_AL_Zeit
      =     #AM_AL_Zeit;
      A     DIX [AR1, P#18.3];  //"DB_NSP".NSP[1].AM_Bad_belegt
      =     #AM_Belegt;
      A     DIX [AR1, P#18.4];  //"DB_NSP".NSP[1].AM_Reset
      =     #Reset;
      A     DIX [AR1, P#2.5];  //"DB_NSP".NSP[1].AL_Ueberlauf
      AN    #Simu;
      =     #AL_Uel;
      A     DIX [AR1, P#2.6];  //"DB_NSP".NSP[1].AL_Niv_min
      AN    #Simu;
      =     #AL_min;
      A     DIX [AR1, P#2.7];  //"DB_NSP".NSP[1].AL_Zeit
      AN    #Simu;
      =     #AL_Zeit;
      A     DIX [AR1, P#19.0];  //"DB_NSP".NSP[1].SprFree
      =     #SPR_free;
      A     DIX [AR1, P#19.1];  //"DB_NSP".NSP[1].NSPFree
      =     #NSP_free;
      A     DIX [AR1, P#19.2];  //"DB_NSP".NSP[1].Warte_NSPT
      =     #Wait_NSPT;

      L     #Pos_Nr;
      +     -1;
      L     "DB_Panel_Posinfo".Leng;
      *D;
      L     "DB_Panel_Posinfo".Offset;
      +D;
      SLD   3;  //Korr. f. Pointer
      T     #Adr_PosInfo_DB;
      LAR2;
      OPN   "DB_Panel_Posinfo";
//x  U     #AL_Zeit
//x  R     DBX [AR2,P#20.0]            //"DB_PC_Posinfo".BAD[1].NS_Auto

      A     DBX [AR2, P#20.0];  //"DB_PC_Posinfo".BAD[1].NS_Auto
      =     #NSP_erlaubt;
      A     DBX [AR2, P#20.1];  //"DB_PC_Posinfo".BAD[1].SR_Auto
      =     #SPR_erlaubt;
      L     DBW [AR2, P#32.0];  //"DB_PC_Posinfo".BAD[1].Zeit_NS
      T     #Zeit_NS;
      L     DBW [AR2, P#24.0];  //"DB_PC_Posinfo".BAD[1].Zeit_SPR
      T     #Zeit_SPR;
      L     DBB [AR2, P#34.0];  //"DB_PC_Posinfo".BAD[1].NS_Kor_Tr
      T     #NS_Kor_Tr;
      L     DBB [AR2, P#35.0];  //"DB_PC_Posinfo".BAD[1].Coun_Kor
      T     #Coun_Kor;
      L     DBW [AR2, P#78.0];
      T     #TestZeit_NS;
      L     DBW [AR2, P#76.0];
      T     #TestZeit_SPR;

      L     #Pos_Nr;
      L     "DB_POS".LENG;
      *D;
      L     "DB_POS".Offset;
      +D;
      SLD   3;
      T     #Adr_Pos_DB;
      LAR2;
      OPN   "DB_POS";
      A     DBX [AR2, P#38.1];  //Leer-WT
      =     #Leer_WT;

      OPN   "DB_POS";
      A     DBX [AR2, P#6.6];  //Hebt
      A(;
      A     "DI_FW_1".OUT.HEBEN_li;
      O     "DI_FW_1".OUT.HEBEN_re;
      );
      =     #Hebt;

      OPN   "DB_POS";
      A     DBX [AR2, P#6.7];  //Senkt
      A(;
      A     "DI_FW_1".OUT.SENKEN_li;
      O     "DI_FW_1".OUT.SENKEN_re;
      );
      =     #Senkt;

      OPN   "DB_POS";
      A     DBX [AR2, P#96.1];  //Bearbeitung
      =     #Bearbeitung;
      A     DBX [AR2, P#96.0];  //Belegt
      =     #belegt;
      A     #belegt;
      AN    #AM_Belegt;
      =     #Eingesetzt;
      AN    #belegt;
      A     #AM_Belegt;
      =     #Ausgehoben;
      L     DBB [AR2, P#5.0];  //akt_FW
      T     #FW_Nr;
      A     DBX [AR2, P#38.0];  //Trommel
      =     #Trommel;
      A     DBX [AR2, P#8.6];  //Spr_off
      A     #Trommel;
      =     #SPR_off;

      L     #Pos_Nr;
      +     -1;
      L     "DB_Panel_OVERVIEW".Leng;
      *D;
      L     "DB_Panel_OVERVIEW".Offset;
      +D;
      SLD   3;
      T     #Adr_Overview_DB;


NETWORK
TITLE = Spritzregister
      A     #Ausgehoben;
      A     #SPR_out;
      O(;
      A     #Eingesetzt;
      A     #SPR_in;
      );
      A     #SPR_Zeit;
      JCN   nIni;

      L     #Zeit_SPR;
      T     #Restzeit_SPR;

nIni: A     "DB_NSP".Test_start;
      R     #SPR_on;
      JC    NV;

      L     #TestZeit_SPR;
      L     0;
      >I;
      =     #SPR_on;
      JC    NV;

      A     "DB_NSP".Test_on;
      O     "DB_NSP".Test_start;
      R     #SPR_erlaubt;

      AN    #SPR_in;
      AN    #SPR_out;
      AN    #SPR_exp;
      ON    #SPR_erlaubt;
      JC    NV;

      A(;
      A(;
      L     "DI_FW_1".ZST.WT_DB_NR_li;
      L     0;
      <>I;
      );
      O(;
      L     "DI_FW_1".ZST.WT_DB_NR_re;
      L     0;
      <>I;
      );
      );
//      U(
//      U(
//      L     "DI_FW_HUB_links".IN.HubInc
//      L     900
//      >D
//      )
//      O(
//      L     "DI_FW_HUB_rechts".IN.HubInc
//      L     900
//      >D
//      )
//      )
      A     "DI_FW_1".ZST.Mittig;
      AN    "DI_FW_1".ZST.HW_mittig;
      AN    "DI_FW_1".ZST.Ofs_mittig;
      =     #Spr_frg;

      AN    #Leer_WT;
      A     #Spr_frg;
      A     #Hebt;
      AN    #SPR_off;
      A     #SPR_out;
      AN    #SPR_Zeit;
      O;
      A     #Senkt;
      A     #Spr_frg;
      A     #SPR_in;
      AN    #SPR_Zeit;
      O;
      AN    #Leer_WT;
      A     #Bearbeitung;
      A     #SPR_exp;
      O;
      A     #ext_Start;
      S     #SPR_on;

      L     #Restzeit_SPR;
      L     0;
      >I;
      A     #SPR_Zeit;
      S     #SPR_on;


NETWORK
TITLE = Allgemeine Freigabe
NV:   A     "DB_NSP".Test_start;
      R     #NS_On;
      JC    Alm;

      L     #TestZeit_NS;
      L     0;
      >I;
      A     #Freigabe;
      =     #NS_On;
      JC    Alm;

      A     "DB_NSP".Test_on;
      R     #NSP_erlaubt;

      AN    #NSP_erlaubt;
      ON    #Freigabe;
      O     #AL_Zeit;
      JC    Alm;


NETWORK
TITLE = Niveau regeln
      AN    #NS_Niv;
      JC    Takt;

      AN    #Niveau_ok;
      S     #NS_On;


NETWORK
TITLE = getaktete NS
Takt: AN    #NST_in;
      AN    #NST_out;
      JC    Alm;

      A     #Ausgehoben;
      A     #NST_out;
      O;
      A     #Eingesetzt;
      A     #NST_in;
      O     #ext_Start;
      JC    Init;
      JU    NS;

Init: AN    #Trommel;
      JC    Ini1;
      L     #NS_Kor_Tr;
      T     #Coun_Kor;
      +     1;
      L     #Zeit_NS;
      *I;
      T     #Restzeit_NS;
      JU    Alm;

Ini1: L     0;
      L     #Coun_Kor;
      ==I;
      JC    Ini3;
      L     1;
      -I;
      JP    Ini2;
      L     0;
Ini2: T     #Coun_Kor;
      JU    Alm;

Ini3: L     #Zeit_NS;
      T     #Restzeit_NS;
      JU    Alm;

NS:   L     #Restzeit_NS;
      L     0;
      >I;
      AN    #Wait_NSPT;
      S     #NS_On;

NETWORK
TITLE = Alarmbehandlung
Alm:  A     "DB_NSP".AMS_new;
      R     #AM_Uel;
      R     #AM_min;
      R     #AM_AL_Zeit;

      A     #Reset;
      R     #Reset;
      R     #AL_Zeit;
      R     "DB_NSP".Reset;

      A     "DB_NSP".Reset;
      S     #Reset;

      L     1;
retA: T     #AL_Nr;
      JL    Alst;
      JU    Ausg;
      JU    Uel;  //1 Überlauf
      JU    min;  //2 MinNiveau
      JU    NSAL;  //3 Nachspeisezeit zu gross
Alst: JU    endA;
//-------------------------------------------
//-------------------------------------------
//Überlauf
Uel:  A     #AL_Uel;
      =     #neu;

      AN    "DB_NSP".noMD_aku_max;
      A     #neu;
      =     #hupen;

      A     #AL_Uel;  //Alarm kommt
      AN    #AM_Uel;
      A     #AL_Send;
      O;
      AN    #AL_Uel;  //Alarm geht
      A     #AM_Uel;
      =     #evt;

      AN    #evt;
      JC    nexA;
      A     #AL_Uel;
      =     #AM_Uel;
      JU    Evt;
//-------------------------------------------
//-------------------------------------------
//Niveau zu niedrig
min:  A     #AL_min;
      =     #neu;

      AN    "DB_NSP".noMD_aku_min;
      A     #neu;
      =     #hupen;

      A     #AL_min;  //Alarm kommt
      AN    #AM_min;
      A     #AL_Send;
      O;
      AN    #AL_min;  //Alarm geht
      A     #AM_min;
      =     #evt;

      AN    #evt;
      JC    nexA;
      A     #AL_min;
      =     #AM_min;
      JU    Evt;
//-------------------------------------------
//-------------------------------------------
//Nachspeisezeit zu gross
NSAL: AN    #NSP_erlaubt;
      R     #AL_Zeit;

      A     #NS_On;
      A     #AL_NS;
      AN    "DB_NSP".noMD_opt_Zeit;
      S     #AL_Zeit;

      A     #AL_Zeit;
      =     #neu;

      AN    "DB_NSP".noMD_aku_Zeit;
      A     #neu;
      =     #hupen;

      A     #AL_Zeit;  //Alarm kommt
      AN    #AM_AL_Zeit;
      O;
      AN    #AL_Zeit;  //Alarm geht
      A     #AM_AL_Zeit;
      =     #evt;

      AN    #evt;
      JC    nexA;
      A     #AL_Zeit;
      =     #AM_AL_Zeit;
      JU    Evt;
//-------------------------------------------
//-------------------------------------------
//Meldung abschicken
Evt:  A     #hupen;
      R     "DB_ANLAGE".config.M_Q_Hupe;

//-------------------------------------------
//-------------------------------------------
//nächster Alarm
nexA: L     #AL_Nr;
      +     1;
      JU    retA;

endA: A     #AL_Uel;
      AN    "DB_NSP".noMD_opt_max;
      O;
      A     #AL_min;
      AN    "DB_NSP".noMD_opt_min;
      JCN   enA1;
      A     #AL_Send;
      S     "DB_NSP".temp_Warn;  //temp.Warnung
enA1: A     #AL_Zeit;
      AN    "DB_NSP".noMD_opt_Zeit;
      JCN   Ausg;
      SET;
      S     "DB_NSP".temp_STM;  //temp.Störung


NETWORK
TITLE = Ausgabe
Ausg: OPN   "DB_Panel_OVERVIEW";
      L     #Adr_Overview_DB;
      LAR2;
      A     #NSP_free;
      JC    nNSP;
      A     #NS_On;
      AN    #AL_Uel;
      =     DBX [AR2, P#20.6];
nNSP: A     #SPR_free;
      JC    nSPR;
      A     #SPR_on;
      AN    #AL_Uel;
      =     DBX [AR2, P#20.7];

nSPR: OPNDI "DB_NSP";
      A     #NS_On;
      AN    #AL_Uel;
      =     DIX [AR1, P#2.3];  //NS_akt
      A     #SPR_on;
      AN    #AL_Uel;
      =     DIX [AR1, P#2.4];  //SP_akt
      A     #AM_min;
      =     DIX [AR1, P#18.0];  //"DB_NSP".NSP[1].AM_AL_min
      A     #AM_Uel;
      =     DIX [AR1, P#18.1];  //"DB_NSP".NSP[1].AM_AL_Uel
      A     #AM_AL_Zeit;
      =     DIX [AR1, P#18.2];  //"DB_NSP".NSP[1].AM_AL_Zeit
      A     #belegt;
      =     DIX [AR1, P#18.3];  //"DB_NSP".NSP[1].AM_Bad_belegt
      A     #Reset;
      =     DIX [AR1, P#18.4];  //"DB_NSP".NSP[1].AM_Reset
      A     #AL_Zeit;
      =     DIX [AR1, P#2.7];  //"DB_NSP".NSP[1].AL_Zeit

      OPN   "DB_Panel_Posinfo";  //Korr. f. Pointer
      L     #Adr_PosInfo_DB;
      LAR2;
      L     #Coun_Kor;
      T     DBB [AR2, P#35.0];  //"DB_PC_Posinfo".BAD[1].Coun_Kor


NETWORK
TITLE = Zeiten zählen
//-------------------------------------------
//keine Sekunde um
      A     "DB_NSP".Takt;
      JC    Sek;

      L     #Restzeit_NS;
      T     DIW [AR1, P#4.0];  //Restzeit
      L     #Restzeit_SPR;
      T     DIW [AR1, P#8.0];  //Restzeit SPR
      JU    next;
//-------------------------------------------
//-------------------------------------------
//Restzeit Nachspeisung
Sek:  L     0;
      L     #Restzeit_NS;
      >=I;
      O     #Wait_NSPT;
      JC    off;
      +     -1;
off:  T     DIW [AR1, P#4.0];  //Restzeit
//-------------------------------------------
//-------------------------------------------
//Testzeit Nachspeisung
      OPN   "DB_Panel_Posinfo";  //Korr. f. Pointer
      L     0;
      L     #TestZeit_NS;
      >=I;
      JC    offN;
      +     -1;
offN: T     DBW [AR2, P#78.0];
//-------------------------------------------
//-------------------------------------------
//Restzeit Spritzen
      L     0;
      L     #Restzeit_SPR;
      >=I;
      JC    ofSR;
      +     -1;
ofSR: T     DIW [AR1, P#8.0];  //Restzeit SPR
//-------------------------------------------
//-------------------------------------------
//Testzeit Spritzregister
      L     0;
      L     #TestZeit_SPR;
      >=I;
      JC    offS;
      +     -1;
offS: T     DBW [AR2, P#76.0];
//-------------------------------------------
//-------------------------------------------
//Alarmverzögerung min/max
      A     #AL_Uel;
      O     #AL_min;
      JC    cntA;
      L     DIW [AR1, P#10.0];  //"DB_NSP".NSP[1].VerzT
      T     DIW [AR1, P#12.0];  //"DB_NSP".NSP[1].RestVerz
      JU    enda_Mig;
cntA: L     0;
      L     DIW [AR1, P#12.0];  //"DB_NSP".NSP[1].RestVerz
      >=I;
      JC    offA;
      +     -1;
offA: T     DIW [AR1, P#12.0];  //"DB_NSP".NSP[1].RestVerz
enda_Mig:NOP   0;
//-------------------------------------------
//-------------------------------------------
//Alarmverzögerung Nachspeisezeit
      L     #TestZeit_NS;
      L     0;
      <=I;
      A     #NS_On;
      AN    #Niveau_ok;
      AN    #AL_Zeit;
      JC    cntN;
      L     DIW [AR1, P#14.0];  // "DB_NSP".NSP[1].VerzNS_AL
      JU    offn_Mig;
cntN: L     0;
      L     DIW [AR1, P#16.0];  //"DB_NSP".NSP[1].RestNS_AL
      >=I;
      JC    offn_Mig;
      +     -1;
offn_Mig:T     DIW [AR1, P#16.0];  //"DB_NSP".NSP[1].RestNS_AL
//-------------------------------------------
      JU    next;

END_FUNCTION

FUNCTION "ToDo" : Void   // FC999, STL
{ S7_Optimized_Access := 'FALSE' }
// stored: AutoNumber false
BEGIN

NETWORK
TITLE = 
      CLR;
      L     0;

END_FUNCTION

FUNCTION "Alarme" : Void
{ S7_Optimized_Access := 'TRUE' }
VERSION : 0.1
   VAR_TEMP 
      i : SInt;
      La_Rot : Bool;
      La_Gelb : Bool;
      La_Blau : Bool;
      Hupe_Quitt_Rot : Bool;
      Hupe_Quitt_Gelb : Bool;
      Hupe_Quitt_Blau : Bool;
      temp_S5Time : S5Time;
      b_TO_Komm_Pnoz : Bool;
      b_VEW_niO : Bool;
   END_VAR


BEGIN
	
	REGION ErrorAcknowledge
	    IF "DB_ANLAGE".IN.Quitt_Err THEN
	        "DB_Alarme".Sammelbit_St := FALSE;
	        "DB_Alarme".auto_aus := FALSE;
	        "DB_Alarme".stop_request := FALSE;
	        FOR #i := 0 TO "Anzahl_Alarm_Woerter" DO
	            "DB_Alarme".MLD[#i] := 0;
	        END_FOR;
	    END_IF;
	END_REGION
	
	REGION Alarms
	    "DB_Alarme".MLD[0].%X0 := "Analogwerte"."LF_CM01.BN01".Drahtbruch;
	    "DB_Alarme".MLD[0].%X1 := "Analogwerte"."LF_CM01.BN01".ungueltig;
	    "DB_Alarme".MLD[0].%X2 := "Analogwerte"."LF_CM01.BN02".Drahtbruch;
	    "DB_Alarme".MLD[0].%X3 := "Analogwerte"."LF_CM01.BN02".ungueltig;
	    "DB_Alarme".MLD[0].%X4 := "Analogwerte"."LF_CM02.BN03".Drahtbruch;
	    "DB_Alarme".MLD[0].%X5 := "Analogwerte"."LF_CM02.BN03".ungueltig;
	    "DB_Alarme".MLD[0].%X6 := "Analogwerte"."LF_CM02.BN04".Drahtbruch;
	    "DB_Alarme".MLD[0].%X7 := "Analogwerte"."LF_CM02.BN04".ungueltig;
	    "DB_Alarme".MLD[0].%X8 := "Analogwerte"."p_HQ01.BP01".Drahtbruch;
	    "DB_Alarme".MLD[0].%X9 := "Analogwerte"."p_HQ01.BP01".ungueltig;
	    "DB_Alarme".MLD[0].%X10 := "Analogwerte"."p_HQ02.BP02".Drahtbruch;
	    "DB_Alarme".MLD[0].%X11 := "Analogwerte"."p_HQ02.BP02".ungueltig;
	    "DB_Alarme".MLD[0].%X12 := "Analogwerte"."p_CM01.BP03".Drahtbruch;
	    "DB_Alarme".MLD[0].%X13 := "Analogwerte"."p_CM01.BP03".ungueltig;
	    "DB_Alarme".MLD[0].%X14 := "Analogwerte"."p_CM01.BP04".Drahtbruch;
	    "DB_Alarme".MLD[0].%X15 := "Analogwerte"."p_CM01.BP04".ungueltig;
	    
	    "DB_Alarme".MLD[1].%X0 := "Analogwerte"."p_CM03.BP05".Drahtbruch;
	    "DB_Alarme".MLD[1].%X1 := "Analogwerte"."p_CM03.BP05".ungueltig;
	    "DB_Alarme".MLD[1].%X2 := "Analogwerte"."p_CM02.BP06".Drahtbruch;
	    "DB_Alarme".MLD[1].%X3 := "Analogwerte"."p_CM02.BP06".ungueltig;
	    "DB_Alarme".MLD[1].%X4 := "Analogwerte"."p_CM02.BP07".Drahtbruch;
	    "DB_Alarme".MLD[1].%X5 := "Analogwerte"."p_CM02.BP07".ungueltig;
	    "DB_Alarme".MLD[1].%X6 := "Analogwerte"."p_CM04.BP08".Drahtbruch;
	    "DB_Alarme".MLD[1].%X7 := "Analogwerte"."p_CM04.BP08".ungueltig;
	    "DB_Alarme".MLD[1].%X8 := "Analogwerte"."p_CM05.BP09".Drahtbruch;
	    "DB_Alarme".MLD[1].%X9 := "Analogwerte"."p_CM05.BP09".ungueltig;
	  
	    "DB_Alarme".MLD[1].%X10 := "Analogwerte"."Dfl_GP01.BF01".Drahtbruch;
	    "DB_Alarme".MLD[1].%X11 := "Analogwerte"."Dfl_GP01.BF01".ungueltig;
	    "DB_Alarme".MLD[1].%X12 := "Analogwerte"."Dfl_GP02.BF02".Drahtbruch;
	    "DB_Alarme".MLD[1].%X13 := "Analogwerte"."Dfl_GP02.BF02".ungueltig;
	   
	    "DB_Alarme".MLD[1].%X14 := "Analogwerte"."Niv_GP01.BL30".Drahtbruch;
	    "DB_Alarme".MLD[1].%X15 := "Analogwerte"."Niv_GP01.BL30".ungueltig AND "E_S_IBC_GP01.BG21";
	    
	    "DB_Alarme".MLD[2].%X0 := "Analogwerte"."Niv_GP02.BL31".Drahtbruch;
	    "DB_Alarme".MLD[2].%X1 := "Analogwerte"."Niv_GP02.BL31".ungueltig AND "E_S_IBC_GP02.BG22";
	    "DB_Alarme".MLD[2].%X2 := "Analogwerte".pH_WR01.Drahtbruch;
	    "DB_Alarme".MLD[2].%X3 := "Analogwerte".pH_WR01.ungueltig;
	    "DB_Alarme".MLD[2].%X4 := "Analogwerte".WZ_1_1.Drahtbruch AND NOT "DI_FW_1".ErrIn.Alarm.NotHalt;
	    "DB_Alarme".MLD[2].%X5 := "Analogwerte".WZ_1_1.ungueltig AND NOT "DI_FW_1".ErrIn.Alarm.NotHalt;
	    "DB_Alarme".MLD[2].%X6 := "Analogwerte".WZ_1_2.Drahtbruch AND NOT "DI_FW_1".ErrIn.Alarm.NotHalt;
	    "DB_Alarme".MLD[2].%X7 := "Analogwerte".WZ_1_2.ungueltig AND NOT "DI_FW_1".ErrIn.Alarm.NotHalt;
	    "DB_Alarme".MLD[2].%X8 := "Analogwerte".WZ_1_3.Drahtbruch AND NOT "DI_FW_1".ErrIn.Alarm.NotHalt;
	    "DB_Alarme".MLD[2].%X9 := "Analogwerte".WZ_1_3.ungueltig AND NOT "DI_FW_1".ErrIn.Alarm.NotHalt;
	    "DB_Alarme".MLD[2].%X10 := "Analogwerte".WZ_1_4.Drahtbruch AND NOT "DI_FW_1".ErrIn.Alarm.NotHalt;
	    "DB_Alarme".MLD[2].%X11 := "Analogwerte".WZ_1_4.ungueltig AND NOT "DI_FW_1".ErrIn.Alarm.NotHalt;
	    "DB_Alarme".MLD[2].%X12 := "Analogwerte".WZ_2_1.Drahtbruch AND NOT "DI_FW_1".ErrIn.Alarm.NotHalt;
	    "DB_Alarme".MLD[2].%X13 := "Analogwerte".WZ_2_1.ungueltig AND NOT "DI_FW_1".ErrIn.Alarm.NotHalt;
	    "DB_Alarme".MLD[2].%X14 := "Analogwerte".WZ_2_2.Drahtbruch AND NOT "DI_FW_1".ErrIn.Alarm.NotHalt;
	    "DB_Alarme".MLD[2].%X15 := "Analogwerte".WZ_2_2.ungueltig AND NOT "DI_FW_1".ErrIn.Alarm.NotHalt;
	    
	    "DB_Alarme".MLD[3].%X0 := "Analogwerte".WZ_2_3.Drahtbruch AND NOT "DI_FW_1".ErrIn.Alarm.NotHalt;
	    "DB_Alarme".MLD[3].%X1 := "Analogwerte".WZ_2_3.ungueltig AND NOT "DI_FW_1".ErrIn.Alarm.NotHalt;
	    "DB_Alarme".MLD[3].%X2 := "Analogwerte".WZ_2_4.Drahtbruch AND NOT "DI_FW_1".ErrIn.Alarm.NotHalt;
	    "DB_Alarme".MLD[3].%X3 := "Analogwerte".WZ_2_4.ungueltig AND NOT "DI_FW_1".ErrIn.Alarm.NotHalt;
	    "DB_Alarme".MLD[3].%X4 := "Analogwerte".Last_1.Drahtbruch AND NOT "DI_FW_1".ErrIn.Alarm.NotHalt;
	    "DB_Alarme".MLD[3].%X5 := "Analogwerte".Last_1.ungueltig AND NOT "DI_FW_1".ErrIn.Alarm.NotHalt;
	    "DB_Alarme".MLD[3].%X6 := "Analogwerte".Last_2.Drahtbruch AND NOT "DI_FW_1".ErrIn.Alarm.NotHalt;
	    "DB_Alarme".MLD[3].%X7 := "Analogwerte".Last_2.ungueltig AND NOT "DI_FW_1".ErrIn.Alarm.NotHalt;
	    "DB_Alarme".MLD[3].%X8 := "DB_Temporaer".Drucksensoren_deaktiviert; //20.01.22
	    "DB_Alarme".MLD[3].%X9 := FALSE;
	    "DB_Alarme".MLD[3].%X10 := FALSE;
	    "DB_Alarme".MLD[3].%X11 := NOT "E_Normal-Vers";
	    "DB_Alarme".MLD[3].%X12 := "DB_NSP".NSP[1].AM_AL_min;
	    "DB_Alarme".MLD[3].%X13 := "DB_NSP".NSP[13].AM_AL_min;
	    "DB_Alarme".MLD[3].%X14 := "DB_NSP".NSP[19].AM_AL_min;
	    "DB_Alarme".MLD[3].%X15 := NOT "E_kein_NB_AblW";
	    
	    "DB_Alarme".MLD[4].%X0 := "Tor".Mld.n_Auto;
	    "DB_Alarme".MLD[4].%X1 := "Tor".Mld.TO_auf;
	    "DB_Alarme".MLD[4].%X2 := "Tor".Mld.TO_zu;
	    "DB_Alarme".MLD[4].%X3 := "Tor".Mld.MSS;
	    "DB_Alarme".MLD[4].%X4 := "Tor".Mld.nok;
	    "DB_Alarme".MLD[4].%X5 := "DB_Schaltuhr".nichtOK;
	    "DB_Alarme".MLD[4].%X6 := "Deckel_CM01".Mld.TO_links_auf;
	    "DB_Alarme".MLD[4].%X7 := "Deckel_CM01".Mld.TO_links_zu;
	    "DB_Alarme".MLD[4].%X8 := "Deckel_CM01".Mld.TO_rechts_auf;
	    "DB_Alarme".MLD[4].%X9 := "Deckel_CM01".Mld.TO_rechts_zu;
	    "DB_Alarme".MLD[4].%X10 := "Deckel_CM01".Mld.Si_24VDC_links;
	    "DB_Alarme".MLD[4].%X11 := "Deckel_CM01".Mld.Si_24VDC_rechts;
	    "DB_Alarme".MLD[4].%X12 := "Deckel_CM01".Mld.n_Auto;
	    "DB_Alarme".MLD[4].%X13 := "Deckel_CM01".Mld.SF_gleich_li_auf;
	    "DB_Alarme".MLD[4].%X14 := "Deckel_CM01".Mld.SF_gleich_li_zu;
	    "DB_Alarme".MLD[4].%X15 := "Deckel_CM01".Mld.SF_gleich_re_auf;
	    
	    "DB_Alarme".MLD[5].%X0 := "Deckel_CM01".Mld.SF_gleich_re_zu;
	    "DB_Alarme".MLD[5].%X1 := "Deckel_CM02".Mld.TO_links_auf;
	    "DB_Alarme".MLD[5].%X2 := "Deckel_CM02".Mld.TO_links_zu;
	    "DB_Alarme".MLD[5].%X3 := "Deckel_CM02".Mld.TO_rechts_auf;
	    "DB_Alarme".MLD[5].%X4 := "Deckel_CM02".Mld.TO_rechts_zu;
	    "DB_Alarme".MLD[5].%X5 := "Deckel_CM02".Mld.Si_24VDC_links;
	    "DB_Alarme".MLD[5].%X6 := "Deckel_CM02".Mld.Si_24VDC_rechts;
	    "DB_Alarme".MLD[5].%X7 := "Deckel_CM02".Mld.n_Auto;
	    "DB_Alarme".MLD[5].%X8 := "Deckel_CM02".Mld.SF_gleich_li_auf;
	    "DB_Alarme".MLD[5].%X9 := "Deckel_CM02".Mld.SF_gleich_li_zu;
	    "DB_Alarme".MLD[5].%X10 := "Deckel_CM02".Mld.SF_gleich_re_auf;
	    "DB_Alarme".MLD[5].%X11 := "Deckel_CM02".Mld.SF_gleich_re_zu;
	    "DB_Alarme".MLD[5].%X12 := NOT "E_Wrn_Gas_ok";
	    "DB_Alarme".MLD[5].%X13 := NOT "E_Al_Gas_ok";
	    "DB_Alarme".MLD[5].%X14 := NOT "E_StrWae_Abluft_ok";
	    "DB_Alarme".MLD[5].%X15 := NOT "DB_PNOZ_IN_Out".In.Abluft_ok OR NOT "E_Frg_AbLW";
	    
	    "DB_Alarme".MLD[6].%X0 := NOT "DB_PNOZ_IN_Out".In.PNOZ_OK AND "DB_PNOZ_IN_Out".In."NH-T_SS_ok" AND "DB_PNOZ_IN_Out".In."NH-T_Filter_ok" AND
	    "DB_PNOZ_IN_Out".In."NH-T_Vers_ok" AND "DB_PNOZ_IN_Out".In."NH-T_Ents_ok" AND "DB_PNOZ_IN_Out".In."NH-T_Vent_ok"  AND "DB_PNOZ_IN_Out".In.NH_MP_ok;
	    
	    "DB_Alarme".MLD[6].%X1 := NOT "DB_PNOZ_IN_Out".In."NH-T_SS_ok";
	    "DB_Alarme".MLD[6].%X2 := NOT "DB_PNOZ_IN_Out".In."NH-T_Filter_ok";
	    "DB_Alarme".MLD[6].%X3 := NOT "DB_PNOZ_IN_Out".In."NH-T_Vers_ok";
	    "DB_Alarme".MLD[6].%X4 := NOT "DB_PNOZ_IN_Out".In."NH-T_Ents_ok";
	    "DB_Alarme".MLD[6].%X5 := NOT "DB_PNOZ_IN_Out".In."NH-T_Vent_ok";
	    "DB_Alarme".MLD[6].%X6 := NOT "DB_PNOZ_IN_Out".In.NH_Frg_TW_QF AND "DB_PNOZ_IN_Out".In.PNOZ_OK;
	    "DB_Alarme".MLD[6].%X7 := NOT "DB_PNOZ_IN_Out".In.NH_MP_ok;
	    "DB_Alarme".MLD[6].%X8 := NOT "DB_PNOZ_IN_Out".In.Tuer_VS_ok;
	    "DB_Alarme".MLD[6].%X9 := NOT "DB_PNOZ_IN_Out".In.Tuer_RS_ok;
	    #temp_S5Time := S_ODT(T_NO := "T-TO-Komm-PNOZ", S := NOT "DB_PNOZ_Comm".RECEIVE.NDR, TV := S5t#1s, Q => #b_TO_Komm_Pnoz);
	    "DB_Alarme".MLD[6].%X10 := #b_TO_Komm_Pnoz;
	    #temp_S5Time := S_ODT(T_NO := "T_VEW_niO", S := NOT "E_VEW_ok", TV := S5t#5s, Q => #b_VEW_niO);
	    "DB_Alarme".MLD[6].%X11 := #b_VEW_niO;
	    "DB_Alarme".MLD[6].%X12 := NOT "E_DL_keine_Warnung" AND "E_DL_min_ok";
	    "DB_Alarme".MLD[6].%X13 := NOT "E_DL_min_ok";
	    "DB_Alarme".MLD[6].%X14 := "E_Not-Strom";
	    "DB_Alarme".MLD[6].%X15 := NOT "E_UeSp_ok";
	    
	    "DB_Alarme".MLD[7].%X0 := NOT "E_Si_230VAC_Bel";
	    "DB_Alarme".MLD[7].%X1 := "FP_CM01.GP01".Mld.GW_p_FP;
	    "DB_Alarme".MLD[7].%X2 := "FP_CM01.GP01".Mld.GW_LF_FP;
	    "DB_Alarme".MLD[7].%X3 := "FP_CM01.GP01".Mld.GW_p_FG;
	    "DB_Alarme".MLD[7].%X4 := "FP_CM01.GP01".Mld.FG_links_nicht_zu;
	    "DB_Alarme".MLD[7].%X5 := "FP_CM01.GP01".Mld.FG_rechts_nicht_zu;
	    "DB_Alarme".MLD[7].%X6 := "FP_CM01.GP01".Mld.Einhausung_nicht_zu;
	    "DB_Alarme".MLD[7].%X7 := "FP_CM01.GP01".Mld.FU_nicht_bereit;
	    "DB_Alarme".MLD[7].%X8 := "FP_CM01.GP01".Mld.FU_Stoerung;
	    "DB_Alarme".MLD[7].%X9 := "FP_CM01.GP01".Mld.FG_Spülen_Ende;
	    "DB_Alarme".MLD[7].%X10 := "FP_CM01.GP01".Mld.n_Auto;
	    "DB_Alarme".MLD[7].%X11 := "FP_CM02.GP04".Mld.Leckage;
	    "DB_Alarme".MLD[7].%X12 := "FP_CM02.GP04".Mld.GW_p_FP;
	    "DB_Alarme".MLD[7].%X13 := "FP_CM02.GP04".Mld.GW_LF_FP;
	    "DB_Alarme".MLD[7].%X14 := "FP_CM02.GP04".Mld.GW_p_FG;
	    "DB_Alarme".MLD[7].%X15 := "FP_CM02.GP04".Mld.FG_links_nicht_zu;
	    
	    "DB_Alarme".MLD[8].%X0 := "FP_CM02.GP04".Mld.FG_rechts_nicht_zu;
	    "DB_Alarme".MLD[8].%X1 := "FP_CM02.GP04".Mld.Einhausung_nicht_zu;
	    "DB_Alarme".MLD[8].%X2 := "FP_CM02.GP04".Mld.FU_nicht_bereit;
	    "DB_Alarme".MLD[8].%X3 := "FP_CM02.GP04".Mld.FU_Stoerung;
	    "DB_Alarme".MLD[8].%X4 := "FP_CM02.GP04".Mld.FG_Spülen_Ende;
	    "DB_Alarme".MLD[8].%X5 := "FP_CM02.GP04".Mld.n_Auto;
	    "DB_Alarme".MLD[8].%X6 := "UP_CM01.GP02".Mld.Niv_TLS;
	    "DB_Alarme".MLD[8].%X7 := "UP_CM01.GP02".Mld.Niv_Ueberlauf;
	    "DB_Alarme".MLD[8].%X8 := "UP_CM01.GP02".Mld.Niv_Sensorfehler;
	    "DB_Alarme".MLD[8].%X9 := "UP_CM01.GP02".Mld.GW_p_UP;
	    "DB_Alarme".MLD[8].%X10 := "UP_CM01.GP02".Mld.GW_LF_UP;
	    "DB_Alarme".MLD[8].%X11 := "UP_CM01.GP02".Mld.FU_nicht_bereit;
	    "DB_Alarme".MLD[8].%X12 := "UP_CM01.GP02".Mld.FU_Stoerung;
	    "DB_Alarme".MLD[8].%X13 := "UP_CM01.GP02".Mld.n_Auto;
	    "DB_Alarme".MLD[8].%X14 := "UP_CM02.GP05".Mld.Niv_TLS;
	    "DB_Alarme".MLD[8].%X15 := "UP_CM02.GP05".Mld.Niv_Ueberlauf;
	    
	    "DB_Alarme".MLD[9].%X0 := "UP_CM02.GP05".Mld.Niv_Sensorfehler;
	    "DB_Alarme".MLD[9].%X1 := "UP_CM02.GP05".Mld.GW_p_UP;
	    "DB_Alarme".MLD[9].%X2 := "UP_CM02.GP05".Mld.GW_LF_UP;
	    "DB_Alarme".MLD[9].%X3 := "UP_CM02.GP05".Mld.FU_nicht_bereit;
	    "DB_Alarme".MLD[9].%X4 := "UP_CM02.GP05".Mld.FU_Stoerung;
	    "DB_Alarme".MLD[9].%X5 := "UP_CM02.GP05".Mld.n_Auto;
	    "DB_Alarme".MLD[9].%X6 := "UP_CM03.GP03".Mld.Niv_TLS;
	    "DB_Alarme".MLD[9].%X7 := "UP_CM03.GP03".Mld.Niv_Sensorfehler;
	    "DB_Alarme".MLD[9].%X8 := "UP_CM03.GP03".Mld.GW_p_UP;
	    "DB_Alarme".MLD[9].%X9 := "UP_CM03.GP03".Mld.FU_nicht_bereit;
	    "DB_Alarme".MLD[9].%X10 := "UP_CM03.GP03".Mld.FU_Stoerung;
	    "DB_Alarme".MLD[9].%X11 := "UP_CM03.GP03".Mld.n_Auto;
	    "DB_Alarme".MLD[9].%X12 := "UP_CM04.GP06".Mld.Niv_TLS;
	    "DB_Alarme".MLD[9].%X13 := "UP_CM04.GP06".Mld.Niv_Sensorfehler;
	    "DB_Alarme".MLD[9].%X14 := "UP_CM04.GP06".Mld.GW_p_UP;
	    "DB_Alarme".MLD[9].%X15 := "UP_CM04.GP06".Mld.FU_nicht_bereit;
	    
	    "DB_Alarme".MLD[10].%X0 := "UP_CM04.GP06".Mld.FU_Stoerung;
	    "DB_Alarme".MLD[10].%X1 := "UP_CM04.GP06".Mld.n_Auto;
	    "DB_Alarme".MLD[10].%X2 := "Pu_CM05.GP11_DB".Mld.MSS;
	    "DB_Alarme".MLD[10].%X3 := "Pu_CM05.GP11_DB".Mld."TLS_CM05.BL03";
	    "DB_Alarme".MLD[10].%X4 := "Pu_CM05.GP11_DB".Mld."Uel_CM05.BL05";
	    "DB_Alarme".MLD[10].%X5 := "Pu_CM05.GP11_DB".Mld.AWA_niO;
	    "DB_Alarme".MLD[10].%X6 := "Pu_CM05.GP11_DB".Mld.keine_Frg_AWA;
	    "DB_Alarme".MLD[10].%X7 := "Pu_CM05.GP11_DB".Mld.Niv_Sensorfehler;
	    "DB_Alarme".MLD[10].%X8 := "Pu_CM05.GP11_DB".Mld.GW_p;
	    "DB_Alarme".MLD[10].%X9 := "Pu_CM05.GP11_DB".Mld.n_Auto;
	    "DB_Alarme".MLD[10].%X10 := "Pu_CL01.GP08".Mld.Leckage;
	    "DB_Alarme".MLD[10].%X11 := "Pu_CL01.GP08".Mld.Niv_Sensorfehler;
	    "DB_Alarme".MLD[10].%X12 := "Pu_CL01.GP08".Mld.n_Auto;
	    "DB_Alarme".MLD[10].%X13 := FALSE;
	    "DB_Alarme".MLD[10].%X14 := "Pu_CL02.GP09".Mld.Leckage;
	    "DB_Alarme".MLD[10].%X15 := "Pu_CL02.GP09".Mld.Niv_Sensorfehler;
	    
	    "DB_Alarme".MLD[11].%X0 := "Pu_CL02.GP09".Mld.n_Auto;
	    "DB_Alarme".MLD[11].%X1 := FALSE;
	    "DB_Alarme".MLD[11].%X2 := "Pu_GP01.GP12".Mld.Leckage;
	    "DB_Alarme".MLD[11].%X3 := "Pu_GP01.GP12".Mld.Niv_Sensorfehler;
	    "DB_Alarme".MLD[11].%X4 := "Pu_GP01.GP12".Mld.n_Auto;
	    "DB_Alarme".MLD[11].%X5 := FALSE;
	    "DB_Alarme".MLD[11].%X6 := "Pu_GP02.GP07".Mld.Leckage;
	    "DB_Alarme".MLD[11].%X7 := "Pu_GP02.GP07".Mld.Niv_Sensorfehler;
	    "DB_Alarme".MLD[11].%X8 := "Pu_GP02.GP07".Mld.n_Auto;
	    "DB_Alarme".MLD[11].%X9 := "Pu_GP02.GP10".Mld.Leckage_Doppelschlauch;
	    "DB_Alarme".MLD[11].%X10 := "Pu_GP01.GP13".Mld.Leckage_Pumpe;
	    "DB_Alarme".MLD[11].%X11 := "Pu_GP01.GP13".Mld.Leckage_PFA_Uebergang;
	    "DB_Alarme".MLD[11].%X12 := "Pu_GP01.GP13".Mld.Leckage_Doppelrohr;
	    "DB_Alarme".MLD[11].%X13 := "Pu_GP01.GP13".Mld.Leckage_Uml_Tunnel;
	    "DB_Alarme".MLD[11].%X14 := "Pu_GP01.GP13".Mld.Niv_Sensorfehler;
	    "DB_Alarme".MLD[11].%X15 := "Pu_GP01.GP13".Mld.GW_Dfl;
	    
	    "DB_Alarme".MLD[12].%X0 := "Pu_GP01.GP13".Mld.Leermeldung;
	    "DB_Alarme".MLD[12].%X1 := "Pu_GP01.GP13".Mld.Vollmeldung;
	    "DB_Alarme".MLD[12].%X2 := "Pu_GP01.GP13".Mld.n_Auto;
	    "DB_Alarme".MLD[12].%X3 := "Pu_GP02.GP10".Mld.Leckage_Pumpe;
	    "DB_Alarme".MLD[12].%X4 := "Pu_GP02.GP10".Mld.Leckage_PFA_Uebergang;
	    "DB_Alarme".MLD[12].%X5 := NOT "E_LS_GP02.BL26";
	    "DB_Alarme".MLD[12].%X6 := NOT "E_LS_GP02.BL33";
	    "DB_Alarme".MLD[12].%X7 := "Pu_GP02.GP10".Mld.Niv_Sensorfehler;
	    "DB_Alarme".MLD[12].%X8 := "Pu_GP02.GP10".Mld.GW_Dfl;
	    "DB_Alarme".MLD[12].%X9 := "Pu_GP02.GP10".Mld.Leermeldung;
	    "DB_Alarme".MLD[12].%X10 := "Pu_GP02.GP10".Mld.Vollmeldung;
	    "DB_Alarme".MLD[12].%X11 := "Pu_GP02.GP10".Mld.n_Auto;
	    "DB_Alarme".MLD[12].%X12 := "Pu_GP01.GP13".Mld.Radarsonde_niO;
	    "DB_Alarme".MLD[12].%X13 := "Pu_GP02.GP10".Mld.Radarsonde_niO;
	    "DB_Alarme".MLD[12].%X14 := "UP_CM01.GP02".Mld.GW_Dfl;
	    "DB_Alarme".MLD[12].%X15 := "UP_CM02.GP05".Mld.GW_Dfl;
	    
	    "DB_Alarme".MLD[13].%X0 := "Ventil_Stati_DB".Mld."TO_auf_CM01.QM18";
	    "DB_Alarme".MLD[13].%X1 := "Ventil_Stati_DB".Mld."TO_zu_CM01.QM18";
	    "DB_Alarme".MLD[13].%X2 := "Ventil_Stati_DB".Mld."SF_CM01.QM18";
	    "DB_Alarme".MLD[13].%X3 := "Ventil_Stati_DB".Mld."TO_auf_CM01.QM19";
	    "DB_Alarme".MLD[13].%X4 := "Ventil_Stati_DB".Mld."TO_zu_CM01.QM19";
	    "DB_Alarme".MLD[13].%X5 := "Ventil_Stati_DB".Mld."SF_CM01.QM19";
	    "DB_Alarme".MLD[13].%X6 := "Ventil_Stati_DB".Mld."TO_auf_CM01.QM20";
	    "DB_Alarme".MLD[13].%X7 := "Ventil_Stati_DB".Mld."TO_zu_CM01.QM20";
	    "DB_Alarme".MLD[13].%X8 := "Ventil_Stati_DB".Mld."SF_CM01.QM20";
	    "DB_Alarme".MLD[13].%X9 := "Ventil_Stati_DB".Mld."TO_auf_CM01.QM25";
	    "DB_Alarme".MLD[13].%X10 := "Ventil_Stati_DB".Mld."TO_zu_CM01.QM25";
	    "DB_Alarme".MLD[13].%X11 := "Ventil_Stati_DB".Mld."SF_CM01.QM25";
	    "DB_Alarme".MLD[13].%X12 := "Ventil_Stati_DB".Mld."TO_auf_CM01.QM26";
	    "DB_Alarme".MLD[13].%X13 := "Ventil_Stati_DB".Mld."TO_zu_CM01.QM26";
	    "DB_Alarme".MLD[13].%X14 := "Ventil_Stati_DB".Mld."SF_CM01.QM26";
	    "DB_Alarme".MLD[13].%X15 := "Ventil_Stati_DB".Mld."TO_auf_CM01.QM27";
	    
	    "DB_Alarme".MLD[14].%X0 := "Ventil_Stati_DB".Mld."TO_zu_CM01.QM27";
	    "DB_Alarme".MLD[14].%X1 := "Ventil_Stati_DB".Mld."SF_CM01.QM27";
	    "DB_Alarme".MLD[14].%X2 := "Ventil_Stati_DB".Mld."TO_auf_CM02.QM55";
	    "DB_Alarme".MLD[14].%X3 := "Ventil_Stati_DB".Mld."TO_zu_CM02.QM55";
	    "DB_Alarme".MLD[14].%X4 := "Ventil_Stati_DB".Mld."SF_CM02.QM55";
	    "DB_Alarme".MLD[14].%X5 := "Ventil_Stati_DB".Mld."TO_auf_CM02.QM56";
	    "DB_Alarme".MLD[14].%X6 := "Ventil_Stati_DB".Mld."TO_zu_CM02.QM56";
	    "DB_Alarme".MLD[14].%X7 := "Ventil_Stati_DB".Mld."SF_CM02.QM56";
	    "DB_Alarme".MLD[14].%X8 := "Ventil_Stati_DB".Mld."TO_auf_CM02.QM57";
	    "DB_Alarme".MLD[14].%X9 := "Ventil_Stati_DB".Mld."TO_zu_CM02.QM57";
	    "DB_Alarme".MLD[14].%X10 := "Ventil_Stati_DB".Mld."SF_CM02.QM57";
	    "DB_Alarme".MLD[14].%X11 := "Ventil_Stati_DB".Mld."TO_auf_CM02.QM62";
	    "DB_Alarme".MLD[14].%X12 := "Ventil_Stati_DB".Mld."TO_zu_CM02.QM62";
	    "DB_Alarme".MLD[14].%X13 := "Ventil_Stati_DB".Mld."SF_CM02.QM62";
	    "DB_Alarme".MLD[14].%X14 := "Ventil_Stati_DB".Mld."TO_auf_CM02.QM63";
	    "DB_Alarme".MLD[14].%X15 := "Ventil_Stati_DB".Mld."TO_zu_CM02.QM63";
	    
	    "DB_Alarme".MLD[15].%X0 := "Ventil_Stati_DB".Mld."SF_CM02.QM63";
	    "DB_Alarme".MLD[15].%X1 := "Ventil_Stati_DB".Mld."TO_auf_CM02.QM64";
	    "DB_Alarme".MLD[15].%X2 := "Ventil_Stati_DB".Mld."TO_zu_CM02.QM64";
	    "DB_Alarme".MLD[15].%X3 := "Ventil_Stati_DB".Mld."SF_CM02.QM64";
	    "DB_Alarme".MLD[15].%X4 := "Ventil_Stati_DB".Mld."TO_auf_HQ01.QM21";
	    "DB_Alarme".MLD[15].%X5 := "Ventil_Stati_DB".Mld."TO_zu_HQ01.QM21";
	    "DB_Alarme".MLD[15].%X6 := "Ventil_Stati_DB".Mld."SF_HQ01.QM21";
	    "DB_Alarme".MLD[15].%X7 := "Ventil_Stati_DB".Mld."TO_auf_HQ01.QM22";
	    "DB_Alarme".MLD[15].%X8 := "Ventil_Stati_DB".Mld."TO_zu_HQ01.QM22";
	    "DB_Alarme".MLD[15].%X9 := "Ventil_Stati_DB".Mld."SF_HQ01.QM22";
	    "DB_Alarme".MLD[15].%X10 := "Ventil_Stati_DB".Mld."TO_auf_HQ01.QM23";
	    "DB_Alarme".MLD[15].%X11 := "Ventil_Stati_DB".Mld."TO_zu_HQ01.QM23";
	    "DB_Alarme".MLD[15].%X12 := "Ventil_Stati_DB".Mld."SF_HQ01.QM23";
	    "DB_Alarme".MLD[15].%X13 := "Ventil_Stati_DB".Mld."TO_auf_HQ01.QM24";
	    "DB_Alarme".MLD[15].%X14 := "Ventil_Stati_DB".Mld."TO_zu_HQ01.QM24";
	    "DB_Alarme".MLD[15].%X15 := "Ventil_Stati_DB".Mld."SF_HQ01.QM24";
	    
	    "DB_Alarme".MLD[16].%X0 := "Ventil_Stati_DB".Mld."TO_auf_HQ01.LV01";
	    "DB_Alarme".MLD[16].%X1 := "Ventil_Stati_DB".Mld."TO_zu_HQ01.LV01";
	    "DB_Alarme".MLD[16].%X2 := "Ventil_Stati_DB".Mld."SF_HQ01.LV01";
	    "DB_Alarme".MLD[16].%X3 := "Ventil_Stati_DB".Mld."TO_auf_HQ02.QM58";
	    "DB_Alarme".MLD[16].%X4 := "Ventil_Stati_DB".Mld."TO_zu_HQ02.QM58";
	    "DB_Alarme".MLD[16].%X5 := "Ventil_Stati_DB".Mld."SF_HQ02.QM58";
	    "DB_Alarme".MLD[16].%X6 := "Ventil_Stati_DB".Mld."TO_auf_HQ02.QM59";
	    "DB_Alarme".MLD[16].%X7 := "Ventil_Stati_DB".Mld."TO_zu_HQ02.QM59";
	    "DB_Alarme".MLD[16].%X8 := "Ventil_Stati_DB".Mld."SF_HQ02.QM59";
	    "DB_Alarme".MLD[16].%X9 := "Ventil_Stati_DB".Mld."TO_auf_HQ02.QM60";
	    "DB_Alarme".MLD[16].%X10 := "Ventil_Stati_DB".Mld."TO_zu_HQ02.QM60";
	    "DB_Alarme".MLD[16].%X11 := "Ventil_Stati_DB".Mld."SF_HQ02.QM60";
	    "DB_Alarme".MLD[16].%X12 := "Ventil_Stati_DB".Mld."TO_auf_HQ02.QM61";
	    "DB_Alarme".MLD[16].%X13 := "Ventil_Stati_DB".Mld."TO_zu_HQ02.QM61";
	    "DB_Alarme".MLD[16].%X14 := "Ventil_Stati_DB".Mld."SF_HQ02.QM61";
	    "DB_Alarme".MLD[16].%X15 := "Ventil_Stati_DB".Mld."TO_auf_HQ02.LV02";
	    
	    "DB_Alarme".MLD[17].%X0 := "Ventil_Stati_DB".Mld."TO_zu_HQ02.LV02";
	    "DB_Alarme".MLD[17].%X1 := "Ventil_Stati_DB".Mld."SF_HQ02.LV02";
	    "DB_Alarme".MLD[17].%X2 := "Ventil_Stati_DB".Mld."TO_auf_CM03.QM33";
	    "DB_Alarme".MLD[17].%X3 := "Ventil_Stati_DB".Mld."TO_zu_CM03.QM33";
	    "DB_Alarme".MLD[17].%X4 := "Ventil_Stati_DB".Mld."SF_CM03.QM33";
	    "DB_Alarme".MLD[17].%X5 := "Ventil_Stati_DB".Mld."TO_auf_CM03.QM34";
	    "DB_Alarme".MLD[17].%X6 := "Ventil_Stati_DB".Mld."TO_zu_CM03.QM34";
	    "DB_Alarme".MLD[17].%X7 := "Ventil_Stati_DB".Mld."SF_CM03.QM34";
	    "DB_Alarme".MLD[17].%X8 := "Ventil_Stati_DB".Mld."TO_auf_CM04.QM72";
	    "DB_Alarme".MLD[17].%X9 := "Ventil_Stati_DB".Mld."TO_zu_CM04.QM72";
	    "DB_Alarme".MLD[17].%X10 := "Ventil_Stati_DB".Mld."SF_CM04.QM72";
	    "DB_Alarme".MLD[17].%X11 := "Ventil_Stati_DB".Mld."TO_auf_CM04.QM73";
	    "DB_Alarme".MLD[17].%X12 := "Ventil_Stati_DB".Mld."TO_zu_CM04.QM73";
	    "DB_Alarme".MLD[17].%X13 := "Ventil_Stati_DB".Mld."SF_CM04.QM73";
	    "DB_Alarme".MLD[17].%X14 := "Ventil_Stati_DB".Mld."TO_auf_CM05.QM61";
	    "DB_Alarme".MLD[17].%X15 := "Ventil_Stati_DB".Mld."TO_zu_CM05.QM61";
	    
